// SIMATIC STEP 7 (V5.x) project COB#1&2_CC#2_07_12_2012
// CPU: CPU 315-2 DP
// CPU: CPU 315-2 DP
// program: S7 Program
// program: S7 Program

SYMBOL_TABLE
"MAIN_POWER_DB"	DB 1	DB 1
"HYDRALIC_DB"	DB 2	DB 2
"TRAVEL_DRIVE_DB"	DB 3	DB 3
"CC_BUNKER_GATE_DB"	DB 4	DB 4
"OVEN_CHARGING_DB"	DB 5	DB 5
"TATA_COMMUNICATION_DB"	DB 6	DB 6	// TATA COMMUNIATION DATA BLOCK
"INSTANCE DB FOR FM350"	DB 7	UDT 2	// INSTANCE DB FOR FM350
"08_LID_MECHANISM_DB"	DB 8	DB 8
"LIFTING_PLATFORM_DB"	DB 9	DB 9	// LIFTING PLATFORM DATA BLOCK
"CMD_FROM_TATA"	DB 10	DB 10	// COMMANDS RECEIVED THROUGH PROFIBUS FROM TATA
"FB_TO_TATA"	DB 11	DB 11	// FEEDBACK TO TATA THROUGH PROFIBUS
"DOOR_EXTRACTOR_DB"	DB 12	DB 12	// DOOR EXTRACTOR MECHANISH DATA BLOCK
"DOOR_CLEANER_DB"	DB 13	DB 13	// DOOR CLEANER MECHANISM DATA BLOCK
"JAMB_CLEANER_DB"	DB 14	DB 14	// JAMB CLEANER MECHANISM DATA BLOCK
"WINCC_DB"	DB 15	DB 15
"COAL_SPILLAGE_SYSTEM_DB"	DB 16	DB 16	// COAL SPILLAGE SYSTEM DATA BLOCK
"SCREW_FEEDER_PF"	DB 17	DB 17	// SCREW FEEDER PROFIBUS
"TRAVEL_PROFIBUS"	DB 18	DB 18
"SF_PROFIBUS"	DB 19	DB 19	// SCREW FEEDER PROFIBUS FINAL
"MAIN_POWER"	FC 1	FC 1	// MAIN POWER ON FUNCTION
"CNT2_CTR"	FC 2	FC 2	// Control counter module FM 350-2
"CNT2_WR"	FC 3	FC 3	// Write data records to FM 350-2
"CNT2_RD"	FC 4	FC 4	// Read data records from FM 350-2
"INPUT_MAPPING"	FC 5	FC 5	// INPUT MAPPING OF ALL INPUT
"OUTPUT_MAPPING"	FC 6	FC 6	// OUTPUT MAPPING OF ALL OUTPUT
"HYDRALIC_FUNCTION"	FC 7	FC 7
"TRAVEL_DRIVE"	FC 8	FC 8
"BUNKER_GATE"	FC 9	FC 9
"OVEN_CHARGING_SF"	FC 10	FC 10	// SCREW FEEDERS OPERATION
"LID_1_MECHANISM"	FC 11	FC 11	// LID MECHANISM OF PUSHER SIDE
"PROFIBUS COMMUNICATION"	FC 12	FC 12	// PROFIBUS COMMUNICATION OF DRIVES
"LID_2_MECHANISM"	FC 13	FC 13	// LID MECHANISM OF MIDDLE SIDE
"LID_3_MECHANISM"	FC 14	FC 14	// LID MECHANISM OF COKE SIDE
"TATA_COMMUNICATION"	FC 21	FC 21	// COMMUNICATION WITH TATA THROUGH PROFIBUS
"SCALE"	FC 105	FC 105	// Scaling Values
"UNSCALE"	FC 106	FC 106	// Unscaling Values
"MAIN_PWR_RDY_FOR_ON"	I 0.0	BOOL	// MAIN POWER READY FOR ON
"MAIN_PWR_ON_FB"	I 0.1	BOOL	// MAIN POWER ON FEEDBACK
"CTRL_PWR_ON_FB"	I 0.2	BOOL	// CONTROL POWER ON FEED BACK
"MAIN_PWR_ON_PB"	I 0.3	BOOL	// MAIN POWER ON PUSH BUTTON
"MAIN_PWR_OFF_PB"	I 0.4	BOOL	// MAIN POWER OFF PUSH BUTTON
"LAMP_TEST_PB"	I 0.5	BOOL	// LAMP TEST PUSH BUTTON CONTROL DESK
"ALRM_ACK_PB"	I 0.6	BOOL	// ALARM ACKNOWLEDGE PUSH BUTTON
"TRA_BYPAS_CMD"	I 0.7	BOOL	// TRAVEL BYPASS COMMAND
"LID_MECH_REP_MODE"	I 1.0	BOOL	// LID MECHANISM REPAIR MODE
"LID_MECH_OPER_MODE"	I 1.1	BOOL	// LID MECHANISM OPERATING MODE
"LID_MECH_MAN_MODE"	I 1.2	BOOL	// LID MECHANISM MANUAL MODE
"LID_MECH_AUTO_MODE"	I 1.3	BOOL	// LID MECHANISM AUTO MODE
"HYD_PUMP_1_RDY_FOR_STA"	I 1.4	BOOL	// HYDRAULIC PUMP 1 READY FOR START
"HYD_PUMP_1_RUN_FB"	I 1.5	BOOL	// HYDRAULIC PUMP 1 RUN FEEDBACK
"HYD_PUMP_1_OVRLD_TRIP"	I 1.6	BOOL	// HYDRAULIC PUMP 1 OVERLOAD TRIP
"TRA_AUTO_MAN_SS"	I 1.7	BOOL	// TRAVEL AUTO / MANUAL SELECTOR SWITCH
"HYD_PUMP_2_RDY_FOR_STA"	I 2.0	BOOL	// HYDRAULIC PUMP 2 READY FOR START
"HYD_PUMP_2_RUN_FB"	I 2.1	BOOL	// HYDRAULIC PUMP 2 RUN FEEDBACK
"HYD_PUMP_2_OVRLD_TRIP"	I 2.2	BOOL	// HYDRAULIC PUMP 2 OVERLOAD TRIP
"CIR_PUMP_RDY_FOR_STA"	I 2.3	BOOL	// CIRCULATION PUMP READY FOR START
"CIR_PUMP_ON_FB"	I 2.4	BOOL	// CIRCULATION PUMP RUNNING FEEDBACK
"CIR_PUMP_OVRLD_TRIP"	I 2.5	BOOL	// CIRCULATION PUMP OVERLOAD TRIP
"COOL_FAN_RDY_FOR_STA"	I 2.6	BOOL	// CIRCULATION PUMP READY FOR START
"PROX_MODE_SEL_SF_1"	I 2.7	BOOL	// PROXIMITY MODE SELECTION SCREW FEEDER 1
"COOL_FAN_RUN_FB"	I 3.0	BOOL	// HYDRAULIC COOLER FAN RUN FEEDBACK
"COOL_FAN_OVRLD_TRIP"	I 3.1	BOOL	// HYDRAULIC COOLER FAN OVERLOAD TRIP
"LID_FRAME_CLR_BYBASS"	I 3.2	BOOL	// LID AND FRAME CLEANER BYPASS INPUT
"SPARE_1"	I 3.3	BOOL
"HYD_CD_LCS_SS"	I 3.5	BOOL	// HYDRAULIC PUMP CD/LCS SELECTOR SWITCH
"HYD_PUMP_1_2_SS"	I 3.6	BOOL	// HYDRAULIC PUMP 1 OR 2 SELECTOR SWITCH
"PROX_MODE_SEL_SF_2"	I 3.7	BOOL	// PROXIMITY MODE SELECTION SCREW FEEDER 2
"PUMP_1_STA_PB"	I 4.0	BOOL	// PUMP 1 START PUSH BUTTON
"PUMP_1_STP_PB"	I 4.1	BOOL	// PUMP 1 STOP PUSH BUTTON
"PUMP_2_STA_PB"	I 4.2	BOOL	// PUMP 2 START PUSH BUTTON
"PUMP_2_STP_PB"	I 4.3	BOOL	// PUMP 2 STOP PUSH BUTTON
"EMER_PB_AT_LCS_41"	I 4.4	BOOL	// EMER_PB_AT_LCS 41
"PUMP_1_STA_PB_LCS"	I 4.5	BOOL	// PUMP 1 START PUSH BUTTON AT LCS
"PUMP_1_STP_PB_LCS"	I 4.6	BOOL	// PUMP 1 STOP PUSH BUTTON AT LCS
"PROX_MODE_SEL_SF_3"	I 4.7	BOOL	// PROXIMITY MODE SELECTION SCREW FEEDER 3
"HYD_PUMP_1_2_SS_LCS"	I 5.0	BOOL	// HYDRAULIC PUMP 1 OR 2 SELECTOR SWITCH LCS
"PUMP_2_STA_PB_LCS"	I 5.1	BOOL	// PUMP 2 START PUSH BUTTON AT LCS
"PUMP_2_STP_PB_LCS"	I 5.2	BOOL	// PUMP 2 STOP PUSH BUTTON AT LCS
"CIR_PUMP_STA_PB"	I 5.3	BOOL	// CIRCULATION PUMP START PUSH BUTTON
"CIR_PUMP_STP_PB"	I 5.4	BOOL	// CIRCULATION PUMP STOP PUSH BUTTON
"COOL_FAN_STA_PB"	I 5.5	BOOL	// COOLLER FAN START PUSH BUTTON
"COOL_FAN_STP_PB"	I 5.6	BOOL	// COOLLER FAN STOP PUSH BUTTON
"LAMP_TEST_AT_HYD_LCS"	I 6.0	BOOL	// LAMP TEST PUSH BUTTON AT HYDRALIC LCCS
"ACCUM_STA_PB"	I 6.1	BOOL	// ACCUMULATOR START PUSH BUTTON
"ACCUM_STP_PB"	I 6.2	BOOL	// ACCUMULATOR STOP PUSH BUTTON
"SPARE_2"	I 6.3	BOOL
"SPARE _3"	I 6.4	BOOL
"SHTOFF_VALVE_LINE_1_OPEN"	I 6.5	BOOL	// SHUTOFF VALVE LINE 1 OPEN
"SHTOFF_VALVE_LINE_2_OPEN"	I 6.6	BOOL	// SHUTOFF VALVE LINE 2 OPEN
"LOW_OIL_TEMP"	I 7.0	BOOL	// HYDRALIC LOW OIL TEMPERATURE FROM (THERM)
"HIGH_OIL_TEMP"	I 7.1	BOOL	// HYDRALIC HIGH OIL TEMPERATURE FROM (THERM)
"MAXI_OIL_TEMP"	I 7.2	BOOL	// HYDRALIC MAXI OIL TEMPERATURE FROM (THERM)
"HYD_LO_OIL_LEV"	I 7.3	BOOL	// HYDRALIC LOW OIL LEVEL FLOAT SWITCH
"HYD_MIN_OIL_LEV"	I 7.4	BOOL	// HYDRALIC MINIMUM OIL LEVEL FLOAT SWITCH
"RET_LIN_FILT_CHOKE"	I 7.5	BOOL	// RETURN LINE FILTER CHOKE
"LOW_OIL_PRES_SW"	I 7.6	BOOL	// LOW OIL PRESSURE SWITCH
"RET_LINE_2_FIL_CHK"	I 7.7	BOOL	// RETURN LINE 2 FILTER CHOKE
"HIGH_OIL_PRES"	I 8.0	BOOL	// HIGH OIL PRESSURE SWITCH
"TRA_GRP_1_RDY_FOR_STA"	I 8.1	BOOL	// TRAVEL GROUP MOTOR 1 READY FOR START
"TRA_GRP_1_MTR_RUN_FB"	I 8.2	BOOL	// TRAVEL GROUP MOTOR 1 RUN FEEDBACK
"TRA_MTR_1_OVRLD_TRIP"	I 8.3	BOOL	// TRAVEL MOTOR 1 OVERLOAD TRIP
"TRA_MTR_2_OVRLD_TRIP"	I 8.4	BOOL	// TRAVEL MOTOR 2 OVERLOAD TRIP
"SIR_RDY_FOR_STA"	I 8.5	BOOL	// SIREN READY FOR START
"SIR_RUN_FB"	I 8.6	BOOL	// SIREN RUNNING FEEDBACK
"HOPPER_STP_PB"	I 8.7	BOOL	// HOPPER GATE STOP PUSH BUTTON
"SIR_OVRLD_TRIP"	I 9.0	BOOL	// SIREN OVERLOAD TRIP
"BRK_1_RDY_FOR_STA"	I 9.1	BOOL	// BRAKE 1 READY FOR START
"BRK_1_RUN_FB"	I 9.2	BOOL	// BRAKE 1 RUN FEEDBACK
"TRA_GRP_2_RDY_FOR_STA"	I 9.3	BOOL	// TRAVEL GROUP MOTOR 2 READY FOR START
"TRA_GRP_2_MTR_RUN_FB"	I 9.4	BOOL	// TRAVEL GROUP MOTOR 2 RUN FEEDBACK
"TRA_MTR_3_OVRLD_TRIP"	I 9.5	BOOL	// TRAVEL MOTOR 3 OVERLOAD TRIP
"TRA_MTR_4_OVRLD_TRIP"	I 9.6	BOOL	// TRAVEL MOTOR 4 OVERLOAD TRIP
"BRK_2_RDY_FOR_STA"	I 10.0	BOOL	// BRAKE 2 READY FOR START
"BRK_2_RUN_FB"	I 10.1	BOOL	// BRAKE 2 RUN FEEDBACK
"TRA_JOY_STK_HME_POS"	I 10.2	BOOL	// TRAVEL JOYSTICK HOME POSITION
"TRA_JOY_STK_FWD_POS"	I 10.3	BOOL	// TRAVEL JOYSTICK FORWARD POSITION
"TRA_JOY_STK_REV_POS"	I 10.4	BOOL	// TRAVEL JOYSTICK REVERSE POSITION
"TRA_JOY_STK_DEAD_MAN_PB"	I 10.5	BOOL	// TRAVEL JOYSTICK DEADMAN PUSH BUTTON
"SPARE_4"	I 10.6	BOOL
"TRA_DRV_1_HW_PF_SS"	I 11.0	BOOL	// TRAVEL DRIVE 1 HARDWARE PROFIBUS SELECTOR SWITCH
"TRA_DRV_1_RUN_FB"	I 11.1	BOOL	// TRAVEL DRIVE 1 RUNING FEEDBACK
"TRA_DRV_1_RDY_FOR_STA"	I 11.2	BOOL	// TRAVEL DRIVE 1 READY FOR START
"TRA_DRV_1_TRIP_FB"	I 11.3	BOOL	// TRAVEL DRIVE 1 TRIP FEED BACK
"TRA_DRV_2_HW_PF_SS"	I 11.4	BOOL	// TRAVEL DRIVE 2 HARDWARE PROFIBUS SELECTOR SWITCH
"TRA_DRV_2_RUN_FB"	I 11.5	BOOL	// TRAVEL DRIVE 2 RUNING FEEDBACK
"TRA_DRV_2_RDY_FOR_STA"	I 11.6	BOOL	// TRAVEL DRIVE 2 READY FOR START
"SPARE_5"	I 11.7	BOOL
"TRA_DRV_2_TRIP_FB"	I 12.0	BOOL	// TRAVEL DRIVE 2 TRIP FEED BACK
"LIMIT_SWITCH_END_FWD_FB"	I 12.1	BOOL	// OVER TRAVEL LIMIT SWITCH
"LONG_TRA_SLOW_SPD"	I 12.2	BOOL	// LONG TRAVEL MAKES SLOW SPEED
"LIMIT_SWITCH_END_REV_FB"	I 12.3	BOOL	// LIMIT SWITCH END REVERSE FEED BACK
"SF_1_HW_PF_SS"	I 12.5	BOOL	// SCREW FEEDER 1 HARDWARE/PROFIBUS SELECTOR SWITCH
"SF_1_RDY_FOR_STA"	I 12.6	BOOL	// SCREW FEEDER 1 READY FOR START
"SPARE _6"	I 12.7	BOOL
"SF_1_RUN_FB"	I 13.0	BOOL	// SCREW FEEDER 1 RUNING FEEDBACK
"SF_1_TRIP_FB"	I 13.1	BOOL	// SCREW FEEDER 1 TRIP FEEDBACK
"SF_2_HW_PF_SS"	I 13.2	BOOL	// SCREW FEEDER 2 HARDWARE/PROFIBUS SELECTOR SWITCH
"SF_2_RDY_FOR_STA"	I 13.3	BOOL	// SCREW FEEDER 2 READY FOR START
"SF_2_RUN_FB"	I 13.4	BOOL	// SCREW FEEDER 2 RUNING FEEDBACK
"SF_2_TRIP_FB"	I 13.5	BOOL	// SCREW FEEDER 2 TRIP FEEDBACK
"SF_3_HW_PF_SS"	I 13.6	BOOL	// SCREW FEEDER 3 HARDWARE/PROFIBUS SELECTOR SWITCH
"SPARE_7"	I 13.7	BOOL
"SF_3_RDY_TO_STA"	I 14.0	BOOL	// SCREW FEEDER 3 READY FOR START
"SF_3_RUN_FB"	I 14.1	BOOL	// SCREW FEEDER 2 RUNING FEEDBACK
"SF_3_TRIP_FB"	I 14.2	BOOL	// SCREW FEEDER 3 TRIP FEEDBACK
"SPARE_8"	I 14.3	BOOL
"DC_POWER_PACK1_ON_CMD"	I 14.4	BOOL
"SF _1_STA_PB"	I 14.5	BOOL	// SCREW FEEDER 1 START PUSH BUTTON
"SF_1_STP_PB"	I 14.6	BOOL	// SCREW FEEDER 1 STOP PUSH BUTTON
"SPARE_9"	I 14.7	BOOL
"SF_1_HIGH_SPD_SEL"	I 15.0	BOOL	// SCREW FEEDER 1 HIGH SPEED SELECTION
"SF_1_LOW_SPD_SEL"	I 15.1	BOOL	// SCREW FEEDER 1 LOW SPEED SELECTION
"SF_2_STA_PB"	I 15.2	BOOL	// SCREW FEEDER 2 START PUSH BUTTON
"SF_2_STP_PB"	I 15.3	BOOL	// SCREW FEEDER 2 STOP PUSH BUTTON
"SF_2_HIGH_SPD_SEL"	I 15.4	BOOL	// SCREW FEEDER 2  HIGH SPEED SELECTION
"SF -2 LOW SPEED SELECT"	I 15.5	BOOL	// SCREW FEEDER 2 LOW SPEED SELECTION
"SF_3_STA_PB"	I 15.6	BOOL	// SCREW FEEDER 3 START PUSH BUTTON
"SPARE_10"	I 15.7	BOOL
"SF_3_STP_PB"	I 16.0	BOOL	// SCREW FEEDER 3 STOP PUSH BUTTON
"SF_3_HI_SPD_SEL"	I 16.1	BOOL	// SCREW FEEDER 3 HIGH SPEED SELECTION
"SF_3_LOW_SPD_SEL"	I 16.2	BOOL	// SCREW FEEDER 3 LOW SPEED SELECTION
"LID_LUT_TANK_RDY_FOR_STA"	I 16.3	BOOL	// LID LUTTING TANK READY FOR START
"LID_LUT_TANK_RUN_FB"	I 16.4	BOOL	// LID LUTTING TANK RUN FEEDBACK
"LID_LUT_TANK_OVRLD_TRIP"	I 16.5	BOOL	// LID LUTTING TANK TRIP FEEDBACK
"LID_LUT_TANK_STA_PB"	I 16.6	BOOL	// LID LUTTING TANK START PUSH BUTTON
"SPARE_11"	I 16.7	BOOL
"LID_LUT_TANK_STP_PB"	I 17.0	BOOL	// LID LUTTING TANK STOP PUSH BUTTON
"MAG_ENER_RDY_FOR_START"	I 17.1	BOOL	// MAGNET ENERGISING READY FOR START
"MAG_1_EMER_FB"	I 17.2	BOOL	// MAGNET 1 ENERGISED FEEDBACK
"MAG_2_EMER_FB"	I 17.3	BOOL	// MAGNET 2 ENERGISED FEEDBACK
"MAG_3_EMER_FB"	I 17.4	BOOL	// MAGNET 2 ENERGISED FEEDBACK
"MAG_RUN_FB"	I 17.5	BOOL	// MAGNET RUNNING FEEDBACK
"MAG 1_STA_PB"	I 17.6	BOOL	// MAGNET 1 START PUSH BUTTON
"SPARE_12"	I 17.7	BOOL
"MAG_1_STP_PB"	I 18.0	BOOL	// MAGNET 1 STOP PUSH BUTTON
"MAG_2_STA_PB"	I 18.1	BOOL	// MAGNET 2 START PUSH BUTTON
"MAG_2_STP_PB"	I 18.2	BOOL	// MAGNET 2 STOP PUSH BUTTON
"MAG_3_STA_PB"	I 18.3	BOOL	// MAGNET 2 START PUSH BUTTON
"MAG_3_STP_PB"	I 18.4	BOOL	// MAGNET 3 STOP PUSH BUTTON
"LID_1_AT_MAG_LS"	I 18.5	BOOL	// LID 1 AT MAGNET LIMIT SWITCH
"LID_2_AT_MAG_LS"	I 18.6	BOOL	// LID 2 AT MAGNET LIMIT SWITCH
"SPARE_13"	I 18.7	BOOL
"LID 3_AT_MAG_LS"	I 19.0	BOOL	// LID 3 AT MAGNET LIMIT SWITCH
"LID_1_OSC_MTR_RDY_STA"	I 19.1	BOOL	// LID 1 OSCILLATION MOTOR READY FOR START
"LID_1_OSC_MTR_RUN_FB"	I 19.2	BOOL	// LID 1 OSCILLATION MOTOR RUN FEEDBACK
"LID_1_OSC_MTR_OLR_TRIP"	I 19.3	BOOL	// LID 1 OSCILLATION MOTOR OVERLOAD TRIP
"LID_2_OSC_MTR_RDY_STA"	I 19.4	BOOL	// LID 2 OSCILLATION MOTOR READY FOR START
"LID_2_OSC_MTR_RUN_FB"	I 19.5	BOOL	// LID 2 OSCILLATION MOTOR RUN FEEDBACK
"LID_2_OSC_MTR_OLR_TRIP"	I 19.6	BOOL	// LID 2 OSCILLATION MOTOR OVERLOAD TRIP
"SPARE14"	I 19.7	BOOL
"LID_3_OSC_MTR_RDY_STA"	I 20.0	BOOL	// LID 3 OSCILLATION MOTOR READY FOR START
"LID_3_OSC_MTR_RUN_FB"	I 20.1	BOOL	// LID 3 OSCILLATION MOTOR RUN FEEDBACK
"LID_3_OSC_MTR_OLR_TRIP"	I 20.2	BOOL	// LID 3 OSCILLATION MOTOR OVERLOAD TRIP FEEDBACK
"LID_1_OSC_MTR_STA_PB"	I 20.3	BOOL	// LID 1 OSCILLATION MOTOR START PUSH BUTTON
"LID_1_OSC_MTR_STP_PB"	I 20.4	BOOL	// LID 1 OSCILLATION MOTOR STOP PUSH BUTTON
"LID_2_OSC_MTR_STA_PB"	I 20.5	BOOL	// LID 2 OSCILLATION MOTOR START PUSH BUTTON
"LID 2_OSC_MTR_STOP_PB"	I 20.6	BOOL	// LID 2 OSCILLATION MOTOR STOP PUSH BUTTON
"SPARE_15"	I 20.7	BOOL
"LID_3_OSC_MTR_STA_PB"	I 21.0	BOOL	// LID 3 OSCILLATION MOTOR START PUSH BUTTON
"LID_3_OSC_MTR_STOP_PB"	I 21.1	BOOL	// LID 3 OSCILLATION MOTOR STOP PUSH BUTTON
"LID_FR_CLN_MTR_1_RDY_STA"	I 21.2	BOOL	// LID FRAME CLEANER MOTOR 1 READY FOR START
"LID_FR_CLNR_MTR_1_RUN_FB"	I 21.3	BOOL	// LID FRAME CLEANER MOTOR 1 RUN FEEDBACK
"LID_FR_CLN_MTR_1_OLR"	I 21.4	BOOL	// LID FRAME CLEANER MOTOR 1 OVERLOAD TRIP
"LID_FR_CLN_MT_2_RDY_STA"	I 21.5	BOOL	// LID FRAME CLEANER MOTOR 2 READY FOR START
"LID_FR_CLN_MTR_2_RUN_FB"	I 21.6	BOOL	// LID FRAME CLEANER MOTOR 2 RUN FEEDBACK
"SPARE_16"	I 21.7	BOOL
"LID_FR_CLN_MTR_2_OLR"	I 22.0	BOOL	// LID FRAME CLEANER MOTOR 2 OVERLOAD TRIP
"LID_FR_CLN_MTR_3_RDY_STA"	I 22.1	BOOL	// LID FRAME CLEANER MOTOR 3 READY FOR START
"LID_FR_CLNR_MTR_3_RUN_FB"	I 22.2	BOOL	// LID FRAME CLEANER MOTOR 3 RUN FEEDBACK
"LID_FR_CLN_MTR_3_OLR"	I 22.3	BOOL	// LID FRAME CLEANER MOTOR 3 OVERLOAD TRIP
"LID_FR_CL_MTR_1_STA_PB"	I 22.4	BOOL	// LID 1 FRAME CLEANER MOTOR START PUSH BUTTON
"LID_FR_CLN_MTR_1_STP_PB"	I 22.5	BOOL	// LID 1 FRAME CLEANER MOTOR STOP PUSH BUTTON
"LID_FR_CL_MT_2_STA_PB"	I 22.6	BOOL	// LID 2 FRAME CLEANER MOTOR START PUSH BUTTON
"SPARE_17"	I 22.7	BOOL
"LID_FR_CLN_MTR_2_STP_PB"	I 23.0	BOOL	// LID 2 FRAME CLEANER MOTOR STOP PUSH BUTTON
"LID_FR_CL_MTR_3_STA_PB"	I 23.1	BOOL	// LID 3 FRAME CLEANER MOTOR START PUSH BUTTON
"LID_FR_CLN_MTR_3_STP_PB"	I 23.2	BOOL	// LID 3 FRAME CLEANER MOTOR STOP PUSH BUTTON
"LID_LIFT_1_CA_FWD_STA"	I 23.3	BOOL	// LID LIFTER 1 CARRIAGE FORWARD START PUSH BUTTON
"LID_LIFT_1_CA_RET_STA"	I 23.4	BOOL	// LID LIFTER 1 CARRIAGE RETRACT START PUSH BUTTON
"LID_LIFT_1_VER_DN_STA"	I 23.5	BOOL	// LID LIFTER 1 VERTICAL DOWN START START PUSH BUTTON
"LID_LIFT_1_VER_UP_STA"	I 23.6	BOOL	// LID LIFTER 1 VERTICAL UP START PUSH BUTTON
"SPARE_18"	I 23.7	BOOL
"LID_FR_CLNR_1_DN_STA"	I 24.0	BOOL	// FRAME CLEANER  1 DOWN START PUSH BUTTON
"LID_FR_CLNR_1_UP_STA"	I 24.1	BOOL	// FRAME CLEANER  1 UP START PUSH BUTTON
"TELESCOPE_1_DOWN_STA"	I 24.2	BOOL	// TELESCOPE 1 DOWN START PUSH BUTTON
"TELESCOPE_1_UP_STA"	I 24.3	BOOL	// TELESCOPE 1 UP START PUSH BUTTON
"SLIDE_GATE_1_CLS_STA"	I 24.4	BOOL	// SLIDE GATE 1 CLOSE START PB
"SLIDE_GATE_1_OPN_STA"	I 24.5	BOOL	// SLIDE GATE 1 OPEN START PB
"SPARE_19"	I 24.6	BOOL
"SPARE_20"	I 24.7	BOOL
"LID_LIFT_1_CAR_FWD_LS"	I 25.0	BOOL	// LID LIFTER 1 CARRIAGE FORWARD LIMIT SWITCH
"LID_LIFT_1_CAR_RET_LS"	I 25.1	BOOL	// LID LIFTER 1 CARRIAGE RETRACT LIMIT SWITCH
"LID_LIFT_1_VER_DN_LS"	I 25.2	BOOL	// LID LIFTER 1 VERTICAL DOWN LIMIT SWITCH
"LID_LIFT_1_VER_UP_LS"	I 25.3	BOOL	// LID LIFTER 1 VERTICAL UP LIMIT SWITCH
"LID_LIFT_1_VER_CLN_LS"	I 25.4	BOOL	// LID LIFTER 1 CLEANING LIMIT SWITCH
"LID_FR_CLNR_1_DN_LS"	I 25.5	BOOL	// LID FRAME CLEANER 1 DOWN  LIMIT SWITCH
"LID_FR_CLNR_1_UP_LS"	I 25.6	BOOL	// LID FRAME CLEANER 1 UP  LIMIT SWITCH
"SPARE_21"	I 25.7	BOOL
"TELES_1_DOWN_LS"	I 26.0	BOOL	// TELESCOPE 1 DOWN  LIMIT SWITCH
"TELES_1_UP_LS"	I 26.1	BOOL	// TELESCOPE 1 UP LIMIT SWITCH
"SLIDE_GATE_1_FWD_LS"	I 26.2	BOOL	// SLIDE GATE 1 FORWARD LIMIT SWITCH
"SLIDE_GATE_1_RET_LS"	I 26.3	BOOL	// SLIDE GATE 1 RETRACT LIMIT SWITCH
"LID_LIFT_2_CAR_FWD_STA"	I 26.5	BOOL	// LID LIFTER 2 CARRIAGE FORWARD START PUSH BUTTOM
"LID_LIFT_2_CAR_RET_STA"	I 26.6	BOOL	// LID LIFTER 2 CARRIAGE RETRACT START PUSH BUTTON
"SPARE_22"	I 26.7	BOOL
"LID_LIFT_2_VER_DN_STA"	I 27.0	BOOL	// LID LIFTER 2 VERTICAL DOWN START START PUSH BUTTON
"LID_LIFT_2_VER_UP_STA"	I 27.1	BOOL	// LID LIFTER 2 VERTICAL UP START PUSH BUTTON
"LID_FR_CLNR_2_DN_STA"	I 27.2	BOOL	// FRAME CLEANER  2 DOWN START PUSH BUTTON
"LID_FR_CLNR_2_UP_STA"	I 27.3	BOOL	// FRAME CLEANER  2 UP START PUSH BUTTON
"TELES_2_DOWN_STA"	I 27.4	BOOL	// TELESCOPE 2 DOWN START PUSH BUTTON
"TELES_2_UP_STA"	I 27.5	BOOL	// TELESCOPE 2 UP START PUSH BUTTON
"SLIDE_GATE_2_CLS_STA"	I 27.6	BOOL	// SLIDE GATE 2  CLOSE START PB
"SPARE_23"	I 27.7	BOOL
"SLIDE_GATE_2_OPN_STA"	I 28.0	BOOL	// SLIDE GATE 2 OPEN START PB
"LID_LIFT_2_CARR_FWD_LS"	I 28.2	BOOL	// LID LIFTER 2 CARRIAGE FORWARD LIMIT SWITCH
"LID_LIFT_2_CARR_RET_LS"	I 28.3	BOOL	// LID LIFTER 2 CARRIAGE RETRACT LIMIT SWITCH
"LID_LIFT_2_VER_DN_LS"	I 28.4	BOOL	// LID LIFTER 2 VERTICAL DOWN LIMIT SWITCH
"LID_LIFT_2_VER_UP_LS"	I 28.5	BOOL	// LID LIFTER 2 VERTICAL UP LIMIT SWITCH
"LID_LIFT_2_CLN_POS_LS"	I 28.6	BOOL	// LID LIFTER 1  CLEANING LIMIT SWITCH
"SPARE_24"	I 28.7	BOOL
"LID_FR_CLNR_2_DOWN_LS"	I 29.0	BOOL	// LID FRAME CLEANER 2 DOWN  LIMIT SWITCH
"LID_FR_CLNR 2_UP_LS"	I 29.1	BOOL	// LID FRAME CLEANER 2 UPLIMIT SWITCH
"TELES_2_DOWN_LS"	I 29.2	BOOL	// TELESCOPE 2 DOWN  LIMIT SWITCH
"TELES_2_UP_LS"	I 29.3	BOOL	// TELESCOPE 2 UP  LIMIT SWITCH
"SLIDE_GATE_2_RET_LS"	I 29.4	BOOL	// SLIDE GATE 2 RETRACT LIMIT SWITCH
"SLIDE_GATE_2_FWD_LS"	I 29.5	BOOL	// SLIDE GATE 2 FORWARD LIMIT SWITCH
"SPARE_25"	I 29.7	BOOL
"LID_LIFT_3_CAR_FWD_STA"	I 30.0	BOOL	// LID LIFTER 3 CARRIAGE FORWARD START PUSH BUTTOM
"LID_LIFT_3_CAR_RET_START"	I 30.1	BOOL	// LID LIFTER 3 CARRIAGE RETRACT START PUSH BUTTOM
"LID_LIFT_3_VER_DN_START"	I 30.2	BOOL	// LID LIFTER 3 VERTICAL UP START PUSH BUTTOM
"LID_LIFT_3_VER_UP_START"	I 30.3	BOOL	// LID LIFTER 3 VERTICAL DOWN START PUSH BUTTOM
"LID_FR_CLNR_3_DN_START"	I 30.4	BOOL	// LID FRAME CLEANER 3 DOWN START PUSH BUTTOM
"LID_FR_CLNR 3_UP_START"	I 30.5	BOOL	// LID FRAME CLEANER 3 UPSTART PUSH BUTTOM
"TELES_3_DN_STA"	I 30.6	BOOL	// TELESCOPE 3 DOWN START PUSH BUTTON
"SPARE_26"	I 30.7	BOOL
"TELES_3_UP_STA"	I 31.0	BOOL	// TELESCOPE 3 UP START PUSH BUTTON
"SLIDE_GATE_3_CLS_STA"	I 31.1	BOOL	// SLIDE GATE 3 CLOSE START PB
"SLIDE_GATE_3_OPN_STA"	I 31.2	BOOL	// SLIDE GATE 3 OPEN START PB
"EMER_STP"	I 31.3	BOOL
"LID_LIFT_3_CAR_FWD_LS"	I 31.4	BOOL	// LID LIFTER 3 CARRIAGE FORWARD LIMIT SWITCH
"LID_LIFT_3_CAR_RET_LS"	I 31.5	BOOL	// LID LIFTER 3 CARRIAGE RETRACT LIMIT SWITCH
"LID_LIFT_3_VER_DN_LS"	I 31.6	BOOL	// LID LIFTER 3 VERTICAL DOWN LIMIT SWITCH
"SPARE_27"	I 31.7	BOOL
"LID_LIFT_3_VER_UP_LS"	I 32.0	BOOL	// LID LIFTER 3 VERTICAL UP LIMIT SWITCH
"LID_LIFT_3_VER_CLN_LS"	I 32.1	BOOL	// LID LIFTER 3 CLEANING LIMIT SWITCH
"LID_FR_CLNR_3_DN_LS"	I 32.2	BOOL	// LID FRAME CLEANER 3 DOWN  LIMIT SWITCH
"LID_FR_CLNR_3_UP_LS"	I 32.3	BOOL	// LID FRAME CLEANER 3 UP  LIMIT SWITCH
"TELES_3_DOWN_LS"	I 32.4	BOOL	// TELESCOPE 3 DOWN  LIMIT SWITCH
"TELES_3_UP_LS"	I 32.5	BOOL	// TELESCOPE 3 UP LIMIT SWITCH
"SLIDE_GATE_3_REV_LS"	I 32.6	BOOL	// SLIDE GATE 3 RETRACT LIMIT SWITCH
"SPARE_28"	I 32.7	BOOL
"SLIDE_GATE_3_FWD_LS"	I 33.0	BOOL	// SLIDE GATE 3 FORWARD LIMIT SWITCH
"LCS_EMERGENCY_STP_PB"	I 33.1	BOOL
"BNKR_GATE_MAN_MODE"	I 33.2	BOOL	// BUNKER GATE MANUAL MODE
"BNKR_GATE_REP_MODE"	I 33.3	BOOL	// BUNKER GATE REPAIR MODE
"BNKR_GATE_1_UP_STA_PB"	I 33.4	BOOL	// BUNKER GATE 1 UP START PUSH BUTTON
"BNKR_GATE_1_DN_STA_PB"	I 33.5	BOOL	// BUNKER GATE 1 DOWN START PUSH BUTTON
"BNKR_GATE_1_OPN_STA_PB"	I 33.6	BOOL	// BUNKER GATE 1 OPEN START PUSH BUTTON
"BUKR_GAT OPATION SEMIAUT"	I 33.7	BOOL	// BUNKER GATE SEMI-AUTO MODE
"BNKR_GATE_1_CL_STA_PB"	I 34.0	BOOL	// BUNKER GATE 1 CLOSE START PUSH BUTTON
"BNKR_GATE_2_UP_STA_PB"	I 34.1	BOOL	// BUNKER GATE 2 UP START PUSH BUTTON
"BNKR_GATE_2_DN_STA_PB"	I 34.2	BOOL	// BUNKER GATE 2 DOWN START PUSH BUTTON
"BNKR_GATE_2_OPN_STA_PB"	I 34.3	BOOL	// BUNKER GATE 2 OPEN START PUSH BUTTON
"BNKR_GATE_2_CL_STA_PB"	I 34.4	BOOL	// BUNKER GATE 2 CLOSE START PUSH BUTTON
"BNKR_GATE_3_UP_STA_PB"	I 34.5	BOOL	// BUNKER GATE 3 UP START PUSH BUTTON
"BNKR_GATE_3_DN_STA_PB"	I 34.6	BOOL	// BUNKER GATE 3 DOWN START PUSH BUTTON
"SPARE_29"	I 34.7	BOOL
"BNKR_GATE_3_OPN_STA_PB"	I 35.0	BOOL	// BUNKER GATE 3 OPEN START PUSH BUTTON
"BNKR_GATE_3_CLS_STA_PB"	I 35.1	BOOL	// BUNKER GATE 3 CLOSE START PUSH BUTTON
"BUKR_GATE_COAL_LD_STA_PB"	I 35.2	BOOL	// BUNKER GATE COAL LOAD START PUSH BUTTON
"BUKR_GATE_COAL_LD_STP_PB"	I 35.3	BOOL	// BUNKER GATE COAL LOAD STOP PUSH BUTTON
"BUNKER_GATE_1_UP_LS"	I 35.4	BOOL	// BUNKER GATE 1 UP LIMIT SWITCH
"BUNKER_GATE_1_DN_LS"	I 35.5	BOOL	// BUNKER GATE 1 DOWN LIMIT SWITCH
"BUNKER_GATE_1_OPEN_LS"	I 35.6	BOOL	// BUNKER GATE 1 OPEN LIMIT SWITCH
"TRVL/SCREW SELECTION"	I 35.7	BOOL	// XXXXXXXXXXXXXXXXXXXXXXXXXXXXX
"BUNKER_GATE_1_CLOSE_LS"	I 36.0	BOOL	// BUNKER GATE 1 CLOSE LIMIT SWITCH
"BUNKER_GATE_1_HOME_LS"	I 36.1	BOOL	// BUNKER GATE 1 HOME LIMIT SWITCH
"BUNKER_GATE_2_UP_LS"	I 36.2	BOOL	// BUNKER GATE 2 UP LIMIT SWITCH
"BUNKER_GATE_2_DN_LS"	I 36.3	BOOL	// BUNKER GATE 2 DOWN LIMIT SWITCH
"BUNKER_GATE_2_OPEN_LS"	I 36.4	BOOL	// BUNKER GATE 2 OPEN LIMIT SWITCH
"BUNKER_GATE_2_CLOSE_LS"	I 36.5	BOOL	// BUNKER GATE 2 CLOSE LIMIT SWITCH
"BUNKER_GATE_2_HOME_LS"	I 36.6	BOOL	// BUNKER GATE 2 HOME LIMIT SWITCH
"LID_FR_CLNR_AUTO_MODE"	I 36.7	BOOL
"BUNKER_GATE_3_UP_LS"	I 37.0	BOOL	// BUNKER GATE 3 UP LIMIT SWITCH
"BUNKER_GATE_3_DN_LS"	I 37.1	BOOL	// BUNKER GATE 3 DOWN LIMIT SWITCH
"BUNKER_GATE_3_OPEN_LS"	I 37.2	BOOL	// BUNKER GATE 3 OPEN LIMIT SWITCH
"BUNKER_GATE_3_CLOSE_LS"	I 37.3	BOOL	// BUNKER GATE 3 CLOSE LIMIT SWITCH
"BUNKER_GATE_3_HOME_LS"	I 37.4	BOOL	// BUNKER GATE 3 HOME LIMIT SWITCH
"HOPPER_1_MAXIMUM_LS"	I 37.5	BOOL	// HOPPER 1 MAXIMUM LIMIT SWITCH
"HOPPER_2_MAXIMUM_LS"	I 37.6	BOOL	// HOPPER 2 MAXIMUM LIMIT SWITCH
"BG_1_HM_STA_PB"	I 37.7	BOOL	// BUNKER GATE 3 HOME START PUSH BUTTON
"HOPPER_3_MAXIMUM_LS"	I 38.0	BOOL	// HOPPER 3  MAXIMUM LIMIT SWITCH
"BNKR_GAT_1_UP_STA_PB_LC"	I 38.1	BOOL	// BUNKER GATE 1 UP START PUSH BUTTON LCS
"BNKR_GAT_1_DN_STA_PB_LC"	I 38.2	BOOL	// BUNKER GATE 1 DOWN START PUSH BUTTON LCS
"BNKR_GAT_1_OPN_STA_PB_LC"	I 38.3	BOOL	// BUNKER GATE 1 OPEN START PUSH BUTTON LCS
"BNKR_GAT_1_CLS_STA_PB_LC"	I 38.4	BOOL	// BUNKER GATE 1 CLOSE  START PUSH BUTTON LCS
"BNKR_GAT_1_HME_STA_PB_LC"	I 38.5	BOOL	// BUNKER GATE 1 HOME START PUSH BUTTON LCS
"BNKR_GAT_2_UP_STA_PB_LC"	I 38.6	BOOL	// BUNKER GATE 2 UP START PUSH BUTTON LCS
"BG_2_HME_STA_PB"	I 38.7	BOOL	// BUNKER 2 HOME START PUSH BUTTON
"BNKR_GAT_2_DN_STA_PB_LC"	I 39.0	BOOL	// BUNKER GATE 2 DOWN START PUSH BUTTON LCS
"BNKR_GAT_2_OPN_STA_PB_LC"	I 39.1	BOOL	// BUNKER GATE 2  OPEN START PUSH BUTTON LCS
"BNKR_GAT_2_CLS_STA_PB_LC"	I 39.2	BOOL	// BUNKER GATE 2 CLOSE START PUSH BUTTON LCS
"BNKR_GAT_2_HM_STA_PB_LC"	I 39.3	BOOL	// BUNKER GATE 2 HOME START PUSH BUTTON LCS
"BNKR_GAT_3_UP_STA_PB_LC"	I 39.4	BOOL	// BUNKER GATE 2 UP START PUSH BUTTON LCS
"BNKR_GAT_3_DN_STA_PB_LC"	I 39.5	BOOL	// BUNKER GATE 3 DOWN START PUSH BUTTON LCS
"BNKR_GAT_3_OPN_STA_PB_LC"	I 39.6	BOOL	// BUNKER GATE 3 OPEN START PUSH BUTTON LCS
"BG_3_HM_STA_PB"	I 39.7	BOOL	// BUNKER GATE 3 HOME START PUSH BUTTON
"BNKR_GAT_3_CL_STA_PB_LC"	I 40.0	BOOL	// BUNKER GATE 3 CLOSE START PUSH BUTTON LCS
"BNKR_GAT3_3_HMSTAP_PB_LC"	I 40.1	BOOL	// BUNKER GATE 3 HOME START PUSH BUTTON LCS
"LCS_91_LAMP_TEST"	I 40.2	BOOL	// LCS-91 LAMP TEST PUSH BUTTON
"LCS_91_EMERGENCY_STOP_PB"	I 40.3	BOOL	// LCS-91 EMERGENCY PUSH BUTTON
"DRIVE1 MACRO_FB"	I 40.4	BOOL
"CD_OR_PC_SEL"	I 40.5	BOOL	// CD OR PC SELECTION
"PREPARE_TO_CHARGE"	I 40.6	BOOL	// PREPARE TO CHARGE
"SF_1_PROXI_CNT_INPUT"	I 40.7	BOOL	// SCREW FEEDER 1 PROXIMITY COUNT INPUT
"OVEN_CHARGING_PB"	I 41.0	BOOL	// OVEN CHARING PB FOR AUTO
"FINISH_CHARGING"	I 41.1	BOOL	// FINISH CHARGING PUSH BUTTON
"LID 1_STOP"	I 41.2	BOOL	// LID -1 STOP PUSH BUTTON CD
"LID 2_STOP"	I 41.3	BOOL	// LID -2 STOP PUSH BUTTON CD
"LID 3_STOP"	I 41.4	BOOL	// LID -3 STOP PUSH BUTTON CD
"LEVEL_START_PB"	I 41.5	BOOL
"SIREN_ON_PB"	I 41.6	BOOL	// SIREN ON PUSH BUTTON
"SF_2_PROXI_CNT_INPUT"	I 41.7	BOOL	// SCREW FEEDER 2 PROXIMITY COUNT INPUT
"QUICK_STOP"	I 42.0	BOOL
"AUTO_POSITION_ACKNOWLEGD"	I 42.1	BOOL
"HPALA_LOW_PRESS_START"	I 42.2	BOOL
"HPALA_FIGH PRESS_START"	I 42.3	BOOL
"BIN_GATE_1_PB"	I 42.4	BOOL	// BIN GATE 1 START PUSH BUTTON
"BIN_GATE_2_PB"	I 42.5	BOOL	// BIN GATE 2 START PUSH BUTTON
"BIN_GATE_3_PB"	I 42.6	BOOL	// BIN GATE 3 START PUSH BUTTON
"SF_3_PROXI_CNT_INPUT"	I 42.7	BOOL	// SCREW FEEDER 3 PROXIMITY COUNT INPUT
"CDC_EMERGENCY_STOP"	I 44.4	BOOL	// CDC EMERGENCY STOP
"ALWAYS_OFF"	M 0.0	BOOL	// ALWAYS OFF BIT
"ALWAYS_ON"	M 0.1	BOOL	// ALWAYS ON BIT
"HALF_SECOND_PULSE_TRAIN"	M 0.2	BOOL	// THIS BIT WILL BE ALWAYS ON FOR 500ms AND OFF FOR 500ms
"ONE_SEC_PULSE"	M 0.3	BOOL	// ONE_RAISING EDGE WILL BE GENERATED PER SECOND
"EMERGENCY_PRESSED"	M 0.4	BOOL	// EMERGENCY PUSH BUTTON PRESSED
"PULSE_GENERATION_BIT"	M 0.5	BOOL	// PULSE GENERATION BIT
"LOW_OIL_TEMPE"	M 45.0	BOOL	// LOW OIL TEMPERATURE
"HOP_1_MAX_LS"	M 66.0	BOOL	// HOPPER 1 MAXIMUM LIMIT SWITCH
"HOP_2_MAX_LS"	M 66.2	BOOL	// HOPPER 2 MAXIMUM LIMIT SWITCH
"HOP_3_MAX_LS_SET"	M 66.4	BOOL	// HOPPER 3 MAXIMUM LIMIT SWITCH SET
"PULSE_20"	M 66.5	BOOL
"SCREW_FEEDER_BYPASS"	M 90.0	BOOL
"TEST_BIT"	M 90.1	BOOL
"TEST_BIT_2"	M 90.2	BOOL
"PULSE_1"	M 90.3	BOOL
"PULSE_2"	M 90.4	BOOL
"TRA_PER_IND_BLINK"	M 90.5	BOOL
"ONE_SECOND_PULSE"	M 162.3	BOOL	// ONE RAISING EDGE PULSE PER SECOND
"PROFIBUS_DRIVE_READ_DATA"	MB 108	BYTE
"PROFIBUS_READ_ERROR_D1"	MW 100	INT
"PROFIBUS_WRITE_ERROR_D1"	MW 102	INT
"PROFIBUS_ADDRESS_1"	MW 104	WORD
"PROFIBUS_ADDRESS_2"	MW 106	WORD
"MAIN_PROGRAM"	OB 1	OB 1	// MAIN PROGRAM - CYCLIC EXECUCTION
"CYCL_FLT"	OB 80	OB 80	// Cycle Time Fault
"I/O_FLT1"	OB 82	OB 82	// I/O Point Fault 1
"OBNL_FLT"	OB 85	OB 85	// OB Not Loaded Fault
"RACK_FLT"	OB 86	OB 86	// Loss of Rack Fault
"COMM_FLT"	OB 87	OB 87	// Communication Fault
"COMPLETE RESTART"	OB 100	OB 100	// Complete Restart
"PROG_ERR"	OB 121	OB 121	// Programming Error
"MOD_ERR"	OB 122	OB 122	// Module Access Error
"TRA_JS_IN_VAL"	PIW 256	WORD
"TRA_DRV_JS_SPD_REF"	PIW 258	INT	// TRAVEL DRIVE JOY STICK SPEED REFERENCE
"TRA_DRV_1_SPD_REF"	PQW 256	INT	// TRAVEL DRIVE 1 SPEED REFERENCE
"TRA_DRV_2_SPD_REF"	PQW 258	INT	// TRAVEL DRIVE 2 SPEED REFERENCE
"MAIN PWR START CMD"	Q 0.0	BOOL	// MAIN POWER ON COMMAND
"MAIN PWR READY IND"	Q 0.1	BOOL	// MAIN POWER READY INDICATION
"CONTROL PWR ON INDICATIO"	Q 0.2	BOOL	// CTRL POWER ON INDICATION
"HYD PMP1 ON CMD"	Q 0.3	BOOL	// HYDRAULIC PUMP 1 ON COMMAND
"HYD PMP2 ON CMD"	Q 0.4	BOOL	// HYDRAULIC PUMP 2 ON COMMAND
"CIR PMP ON CMD"	Q 0.5	BOOL	// HYDRAULIC CIRCULATION PUMP ON COMMAND
"COOL FAN ON CMD"	Q 0.6	BOOL	// HYDRAULIC COOLER FAN ON COMMAND
"PRE RELIF VALVE_1 ON CMD"	Q 0.7	BOOL	// PRESSURE RELIEF VALVE ON COMMAND
"SPARE OP 1"	Q 1.0	BOOL
"HYD SYSTEM READY IND"	Q 1.1	BOOL	// HYDRAULIC SYSTEM READY INDICATION
"PUMP1 ON IND CD"	Q 1.2	BOOL	// PUMP 1 ON INDICATION CD
"PUMP2 ON IND CD"	Q 1.3	BOOL	// PUMP 2 ON INDICATION CD
"PUMP1 ON IND LCS"	Q 1.4	BOOL	// PUMP 1 ON INDICATION LCS
"PUMP2 ON IND LCS"	Q 1.5	BOOL	// PUMP 2 ON INDICATION LCS
"CIRC PMP ON IND_LCS"	Q 1.6	BOOL	// CIRCULATION PUMP  ON INDICATION LCS
"SF1 BCD1_3"	Q 1.7	BOOL
"COOL FAN ON IND_LCS"	Q 2.0	BOOL	// COOLER FAN  ON INDICATION LCS
"LOCAL ON IND"	Q 2.1	BOOL	// LOCAL SELECTION ON INDICATION LCS
"HIGH TEMP ON IND_LCS"	Q 2.2	BOOL	// HIGH TEMPERATURE ON INDICATION LCS
"LOWER OIL LVL ON IND_LCS"	Q 2.3	BOOL	// LOWER OIL LEVEL INDICATON LCS
"FILTER CHOHE ON IND_LCS"	Q 2.4	BOOL	// FILTER CHOKE ON INDICATION LCS
"ACCUM_IN_OPER_LCS"	Q 2.5	BOOL	// ACCUMULATOR ON INDICATION LCS
"HEAT_ON_IND_LCS"	Q 2.6	BOOL	// HEATER ON INDICATION LCS
"LOW OIL TEMPERATURE"	Q 2.7	BOOL	// LOWER OIL TEMPERATURE  INDICATON LCS
"TRA GROUP1 ON CMD"	Q 3.0	BOOL
"TRA GROUP2 ON CMD"	Q 3.1	BOOL
"SIREN ON CMD"	Q 3.2	BOOL
"BRAKE ON CMD1"	Q 3.3	BOOL
"BRAKE ON CMD2"	Q 3.4	BOOL
"AUDIO_VISUAL_ALRM_ON_CMD"	Q 3.5	BOOL
"TRA_DRV_FWD"	Q 3.6	BOOL
"TRA_AUD_VIS"	Q 3.7	BOOL	// TRAVEL AUDIO VISUAL SIREN
"TRA_DRV_REV"	Q 4.0	BOOL
"LOGIC I/P 1 TO TR DRIVE"	Q 4.1	BOOL
"LOGIC I/P 2 TO TR DRIVE"	Q 4.2	BOOL
"LOGIC I/P 3 TO TR DRIVE"	Q 4.3	BOOL
"TRA PERMISSION IND"	Q 4.4	BOOL
"TRVL D1 FWD ON CMD"	Q 4.5	BOOL
"TRVL D1 REV ON CMD"	Q 4.6	BOOL
"SPARE 53"	Q 4.7	BOOL
"TRVL D2 FWD ON CMD"	Q 5.0	BOOL
"TRVL D2 REV ON CMD"	Q 5.1	BOOL
"SF -1 HIGH SPEED CMD"	Q 5.2	BOOL
"SF -1 LOW SPEED CMD"	Q 5.3	BOOL
"SF -2 HIGH SPEED CMD"	Q 5.4	BOOL
"SF -2 LOW SPEED CMD"	Q 5.5	BOOL
"SF -3 HIGH SPEED CMD"	Q 5.6	BOOL
"SPARE 52"	Q 5.7	BOOL
"SF -3 LOW SPEED CMD"	Q 6.0	BOOL
"SF -1 ON IND"	Q 6.1	BOOL
"SF -2 ON IND"	Q 6.2	BOOL
"SF -3 ON IND"	Q 6.3	BOOL
"LID LUT TANK ON CMD"	Q 6.4	BOOL
"LID LUT TANK ON IND"	Q 6.5	BOOL
"MAG1 ON CMD"	Q 6.6	BOOL
"BOSTER_CONT_1_ON_CMD"	Q 6.7	BOOL
"MAG2 ON CMD"	Q 7.0	BOOL
"MAG3 ON CMD"	Q 7.1	BOOL
"MAGNET ON CMD"	Q 7.2	BOOL
"MAG1 ON IND"	Q 7.3	BOOL
"MAG2 ON IND"	Q 7.4	BOOL
"MAG3 ON IND"	Q 7.5	BOOL
"LID1 AT MAGNET ON IND"	Q 7.6	BOOL
"BOSTER_CONT_2_ON_CMD"	Q 7.7	BOOL
"LID2 AT MAGNET ON IND"	Q 8.0	BOOL
"LID3 AT MAGNET ON IND"	Q 8.1	BOOL
"LID OSCILLATION1 ON CMD"	Q 8.2	BOOL
"LID OSCILLATION2 ON CMD"	Q 8.3	BOOL
"LID OSCILLATION3 ON CMD"	Q 8.4	BOOL
"LID OSCILLATION1 ON IND"	Q 8.5	BOOL
"LID OSCILLATION2 ON IND"	Q 8.6	BOOL
"BOSTER_CONT_3_ON_CMD"	Q 8.7	BOOL
"LID OSCILLATION3 ON IND"	Q 9.0	BOOL
"LID FR CLEANER1 ON CMD"	Q 9.1	BOOL
"LID FR CLEANER2 ON CMD"	Q 9.2	BOOL
"LID FR CLEANER3 ON CMD"	Q 9.3	BOOL
"LID FR CLEANER1 ON IND"	Q 9.4	BOOL
"LID FR CLEANER2 ON IND"	Q 9.5	BOOL
"LID FR CLEANER3 ON IND"	Q 9.6	BOOL
"SF2 BCD1_4"	Q 9.7	BOOL
"LID LIFT1 CARGE FWD CMD"	Q 10.0	BOOL
"LID LIFT1 CARGE REV CMD"	Q 10.1	BOOL
"LID LIFT1 VERT DWN CMD"	Q 10.2	BOOL
"LID LIFT1 VERT UP CMD"	Q 10.3	BOOL
"LID FR CLEANER1 DOWN CMD"	Q 10.4	BOOL
"LID FR CLEANER1 UP CMD"	Q 10.5	BOOL
"TELESCOPE1 DOWN CMD"	Q 10.6	BOOL
"SF2 BCD1_6"	Q 10.7	BOOL
"TELESCOPE1 UP CMD"	Q 11.0	BOOL
"SLIDE GATE1 CLOSE CMD"	Q 11.1	BOOL
"SLIDE GATE1 OPEN CMD"	Q 11.2	BOOL
"LID LIFT1 CARGE FWD IND"	Q 11.4	BOOL
"LID LIFT1 CARGE REV IND"	Q 11.5	BOOL
"LID LIFT1 VERT DWN IND"	Q 11.6	BOOL
"SF2 BCD1_8"	Q 11.7	BOOL
"LID LIFT1 VERT UP IND"	Q 12.0	BOOL
"LID LIFT1 CLENR POS IND"	Q 12.1	BOOL
"LID FR CLEANER1 DOWN IND"	Q 12.2	BOOL
"LID FR CLEANER1 UP IND"	Q 12.3	BOOL
"TELESCOPE1 DOWN IND"	Q 12.4	BOOL
"TELESCOPE1 UP IND"	Q 12.5	BOOL
"SLIDE GATE1 CLOSE IND"	Q 12.6	BOOL
"SF3 BCD1_1"	Q 12.7	BOOL
"SLIDE GATE1 OPEN IND"	Q 13.0	BOOL
"LID LIFT2 CARGE FWD CMD"	Q 13.2	BOOL
"LID LIFT2 CARGE REV CMD"	Q 13.3	BOOL
"LID LIFT2 VERT DOWN CMD"	Q 13.4	BOOL
"LID LIFT2 VERT UP CMD"	Q 13.5	BOOL
"LID FR CLENR2 DOWN CMD"	Q 13.6	BOOL
"SF3 BCD1_3"	Q 13.7	BOOL
"LID FR CLENR2 UP CMD"	Q 14.0	BOOL
"TELESCOPE2 DOWN CMD"	Q 14.1	BOOL
"TELESCOPE2 UP CMD"	Q 14.2	BOOL
"SLIDE GATE2 CLOSE CMD"	Q 14.3	BOOL
"SLIDE GATE2 OPEN CMD"	Q 14.4	BOOL
"SPARE OUTPUT 6"	Q 14.5	BOOL
"LID LIFT2 CARGE FWD IND"	Q 14.6	BOOL
"SF3 BCD1_4"	Q 14.7	BOOL
"LID LIFT2 CARGE REV IND"	Q 15.0	BOOL
"LID LIFT2 VERT DWN IND"	Q 15.1	BOOL
"LID LIFT2 VERT UP IND"	Q 15.2	BOOL
"LID LIFT2 CLENR POS IND"	Q 15.3	BOOL
"LID FR CLENR2 DOWN IND"	Q 15.4	BOOL
"LID FR CLENR2 UP IND"	Q 15.5	BOOL
"TELESCOPE2 DOWN IND"	Q 15.6	BOOL
"SF3 BCD1_6"	Q 15.7	BOOL
"TELESCOPE2 UP IND"	Q 16.0	BOOL
"SLIDE GATE2 CLOSE IND"	Q 16.1	BOOL
"SLIDE GATE2 OPEN IND"	Q 16.2	BOOL
"LID LIFT3 CARGE FWD CMD"	Q 16.4	BOOL
"LID LIFT3 CARGE REV CMD"	Q 16.5	BOOL
"LID LIFT3 VERT DWN CMD"	Q 16.6	BOOL
"SF3 BCD1_8"	Q 16.7	BOOL
"LID LIFT3 VERT UP CMD"	Q 17.0	BOOL
"LID FR CLENR3 DOWN CMD"	Q 17.1	BOOL
"LID FR CLENR3 UP CMD"	Q 17.2	BOOL
"TELESCOPE3 DOWN CMD"	Q 17.3	BOOL
"TELESCOPE3 UP CMD"	Q 17.4	BOOL
"SLIDE GATE3 CLOSE CMD"	Q 17.5	BOOL
"SLIDE GATE3 OPEN CMD"	Q 17.6	BOOL
"SPARE OUTPUT1"	Q 17.7	BOOL
"LID LIFT3 CARGE FWD IND"	Q 18.1	BOOL
"LID LIFT3 CARGE REV IND"	Q 18.2	BOOL
"LID LIFT3 VERT DWN IND"	Q 18.3	BOOL
"LID LIFT3 VERT UP IND"	Q 18.4	BOOL
"LID LIFT3 CLENR POS IND"	Q 18.5	BOOL
"LID FR CLENR3 DOWN IND"	Q 18.6	BOOL
"SPARE OUTPUT3"	Q 18.7	BOOL
"LID FR CLENR3 UP IND"	Q 19.0	BOOL
"TELESCOPE3 DOWN IND"	Q 19.1	BOOL
"TELESCOPE3 UP IND"	Q 19.2	BOOL
"SLIDE GATE3 CLOSE IND"	Q 19.3	BOOL
"SLIDE GATE3 OPEN IND"	Q 19.4	BOOL
"SPARE OUTPUT7"	Q 19.5	BOOL
"BUNKER GATE1 UP CMD"	Q 19.6	BOOL
"SPARE OUTPUT9"	Q 19.7	BOOL
"BUNKER GATE1 DOWN CMD"	Q 20.0	BOOL
"BUNKER GATE1 OPEN CMD"	Q 20.1	BOOL
"BUNKER GATE1 CLOSE CMD"	Q 20.2	BOOL
"BUNKER GATE2 UP CMD"	Q 20.3	BOOL
"BUNKER GATE2 DOWN CMD"	Q 20.4	BOOL
"BUNKER GATE2 CLOSE CMD"	Q 20.5	BOOL
"BUNKER GATE2 OPEN CMD"	Q 20.6	BOOL
"SPARE OUTPUT17"	Q 20.7	BOOL
"BUNKER GATE3 UP CMD"	Q 21.0	BOOL
"BUNKER GATE3 DOWN CMD"	Q 21.1	BOOL
"BUNKER GATE3 CLOSE CMD"	Q 21.2	BOOL
"BUNKER GATE3 OPEN CMD"	Q 21.3	BOOL
"BUNKER GATE COAL LOD IND"	Q 21.4	BOOL
"LOADING PROGRESS IND"	Q 21.5	BOOL
"BUNKER GATE1 UP IND"	Q 21.6	BOOL
"SPARE OUTPUT18"	Q 21.7	BOOL
"BUNKER GATE1 DOWN IND"	Q 22.0	BOOL
"BUNKER GATE1 OPEN IND"	Q 22.1	BOOL
"BUNKER GATE1 CL0SE IND"	Q 22.2	BOOL
"BUNKER GATE1 HOME IND"	Q 22.3	BOOL
"BUNKER GATE2 UP IND"	Q 22.4	BOOL
"BUNKER GATE2 DN IND"	Q 22.5	BOOL
"BUNKER GATE2 OPEN IND"	Q 22.6	BOOL
"SPARE OUTPUT19"	Q 22.7	BOOL
"BUNKER GATE2 CL0SE IND"	Q 23.0	BOOL
"BUNKER GATE2 HOME IND"	Q 23.1	BOOL
"BUNKER GATE3 UP IND"	Q 23.2	BOOL
"BUNKER GATE3 DOWN IND"	Q 23.3	BOOL
"BUNKER GATE3 OPEN IND"	Q 23.4	BOOL
"BUNKER GATE3 CL0SE IND"	Q 23.5	BOOL
"BUNKER GATE3 HOME IND"	Q 23.6	BOOL
"SPARE OUTPUT20"	Q 23.7	BOOL
"HOPPER1 MAXIMUM IND"	Q 24.0	BOOL
"HOPPER2 MAXIMUM IND"	Q 24.1	BOOL
"HOPPER3 MAXIMUM IND"	Q 24.2	BOOL
"BUNKER GATE 1 UP IND LCS"	Q 24.3	BOOL
"BUNKER GATE 1 DN IND LCS"	Q 24.4	BOOL
"BUNKER GATE 1 OP IND LCS"	Q 24.5	BOOL
"BUNKER GATE 1 CL IND LCS"	Q 24.6	BOOL
"SPARE OUTPUT21"	Q 24.7	BOOL
"BUNKER GATE 1 HM IND LCS"	Q 25.0	BOOL
"BUNKER GATE 2 UP IND LCS"	Q 25.1	BOOL
"BUNKER GATE 2 DN IND LCS"	Q 25.2	BOOL
"BUNKER GATE 2 OP IND LCS"	Q 25.3	BOOL
"BUNKER GATE 2 CL IND LCS"	Q 25.4	BOOL
"BUNKER GATE 2 HM IND LCS"	Q 25.5	BOOL
"BUNKER GATE 3 UP IND LCS"	Q 25.6	BOOL
"SPARE OUTPUT22"	Q 25.7	BOOL
"BUNKER GATE 3 DN IND LCS"	Q 26.0	BOOL
"BUNKER GATE 3 OP IND LCS"	Q 26.1	BOOL
"BUNKER GATE 3 CL IND LCS"	Q 26.2	BOOL
"BUNKER GATE 3 HM IND LCS"	Q 26.3	BOOL
"HOPPER 1 MAXI INDI LCS"	Q 26.4	BOOL
"HOPPER 2 MAXI INDI LCS"	Q 26.5	BOOL
"HOPPER 3 MAXI INDI LCS"	Q 26.6	BOOL
"SPARE OUTPUT25"	Q 26.7	BOOL
"LOCAL SELECTION INDICATI"	Q 27.0	BOOL
"CHARGNG PERMISSION IND"	Q 27.1	BOOL
"CHARGING COMPLETED IND"	Q 27.2	BOOL
"PREPARE TO CHARGE IND"	Q 27.3	BOOL
"OVEN CHARGING IND"	Q 27.4	BOOL
"FINISH CHARGING IND"	Q 27.5	BOOL
"LID 1 PROGRESS IND"	Q 27.6	BOOL
"SPARE OUTPUT29"	Q 27.7	BOOL
"LID 2 PROGRESS IND"	Q 28.0	BOOL
"LID 3 PROGRESS IND"	Q 28.1	BOOL
"LEVEL START"	Q 28.2	BOOL
"HPALA LOP PRESS ON IND"	Q 28.3	BOOL
"PRESSURE RELIEF VALVE 2"	Q 28.4	BOOL
"ACC ON CMD"	Q 28.5	BOOL
"DPRD_DAT"	SFC 14	SFC 14	// Read Consistent Data of a Standard DP Slave
"DPWR_DAT"	SFC 15	SFC 15	// Write Consistent Data to a Standard DP Slave
"BLKMOV"	SFC 20	SFC 20	// Copy Variables
"CREAT_DB"	SFC 22	SFC 22	// Create Data Block
"WR_REC"	SFC 58	SFC 58	// Write Data Record
"RD_REC"	SFC 59	SFC 59	// Read a Data Record
"AUTO_VER_UP_1_DEL"	T 10	TIMER	// VERTICAL UP 1 TIME DELAY AFTER MAGNET OFF
"AUTO_OSC_MTR_ON_OVR"	T 12	TIMER	// AUTO OSCILLATION MOTOR ON TIMER
"BOOSTER_1_OFF_TIMER"	T 13	TIMER	// BOOSTER 1 OFF TIMER
"BOSTER_CONT_2_OFF_TIMER"	T 14	TIMER
"LID_OSC_FB_FLT_TIMER"	T 16	TIMER
"LID_3_OSC_FB_FLT"	T 18	TIMER	// LID OSCILLATION 3 FEEDBACK FLT
"AUTO_OSC_MTR_2_ON_OVR"	T 20	TIMER	// OSCILLATION MOTOR 1 ON OVER
"SF_1_ON_DEL_TIMER"	T 27	TIMER	// SCREW FEEDER 1 ON DELAY TIMER
"SF_2_ON_DEL_TIMER"	T 28	TIMER	// SCREW FEEDER 2 ON DELAY TIMER
"LID_2_VER_UP_TIM_DEL"	T 29	TIMER	// LID 2 VERTICAL UP TIME DELAY AFTER MAGNET OFF
"AUTO_OSC_MTR_3_ON_OVR"	T 30	TIMER	// AUTO OSCILLATION MOTOR 3  ON OVER
"LID_3_VER_UP_TIM_DEL"	T 31	TIMER	// LID 3 VERTICAL UP DELAY AFTER MAGNET OFF
"LID_FR_CLN_MTR_1_OFF_TIM"	T 32	TIMER	// LID FRAME CLEANER MOTOR 1 OFF TIMER
"LID_FRM_CLNR_UP_DEL_TIM"	T 33	TIMER	// LID FRAME CLEANER UP DELAY TIMER
"LID_FRM_CLN_2_UP_DEL_TIM"	T 34	TIMER	// LID FRAME CLEANER 2 MOTOR OFF TIMER
"LID_FRM_CLN_2_STOP_TIM"	T 35	TIMER
"LID_FRM_CLN_UP_DEL_TIM"	T 36	TIMER	// LID FRAME CLEANER UP DELAY TIMER
"LID_FR_CLN_MTR_3_OFF_TIM"	T 37	TIMER	// LID FRAME CLEANER MOTOR 3 OFF TIMER
"BG_1_MAX_LS_CLS_TIM"	T 38	TIMER	// BUNKER GATE 1 MAXIMUM LIMIT SWITCH REACHED
"BG_2_MAX_LS_CLS_TIM"	T 39	TIMER	// BUNKER GATE 2  MAXIMUM LIMIT SWITCH REACHED
"BG_3_MAX_LS_CLS_TIM"	T 40	TIMER	// BUNKER GATE 3  MAXIMUM LIMIT SWITCH REACHED
"PREPARE_CHARGE"	UDT 1	UDT 1
"SCREW_FEEDER"	UDT 2	UDT 2
"FINISH_CHARGE"	UDT 3	UDT 3
"SCREW_FEEDER_SP"	VAT 1		// SCREW FEEDER SET POINTS
"VAT_2"	VAT 2		// OUTPUT_LIST
"VAT_32"	VAT 3	
"PUSHER_RAM_ENCODER"	VAT 4	
"DE_CTRL_SEL_FORCING"	VAT 5	
END_SYMBOL_TABLE

TYPE "PREPARE_CHARGE"	// UDT 1
VERSION : 0.1
  STRUCT
   STEP1 : BOOL ;	//LID LIFTER CAR TRAVEL FWD OVER
   STEP2 : BOOL ;	//LID LIFTER VERT DOWN OVER
   STEP3 : BOOL ;	//LID MAGNET ON FB
   STEP4 : BOOL ;	//LID OSC MOTOR OPRN OVER
   STEP5 : BOOL ;	//LID LIFTER VERT UP OVER
   STEP6 : BOOL ;	//LID LIFTER CAR TRAVEL REV OVER
   STEP7 : BOOL ;	//LID FRAME CLEANER DOWN OVER
   STEP8 : BOOL ;	//LID LIFTER CAR TRAVEL FWD OVER
   STEP9 : BOOL ;	//LID LIFTER VERT DOWN FOR CLN POS OVER
   STEP10 : BOOL ;	//LID CLEANER MOTOR OPRN OVER
   STEP11 : BOOL ;	//LID LIFTER VERT UP FROM CLN POS OVER
   STEP12 : BOOL ;	//LID LIFTER CAR TRAVEL REV OVER
   STEP13 : BOOL ;	//LID FRAME CLEANER UP OVER
   STEP14 : BOOL ;	//TELESCOPE DOWN OVER
   STEP15 : BOOL ;	//LID CLEANER BYPASS ENABLED
   STEP16 : BOOL ;	//LID OSC MOTOR TIME OVER
   STEP17 : BOOL ;	//LID CLEANER MOTOR TIME OVER
   STEP19 : BOOL ;	//PREPARE CHARGE OPERATION COMPLETED
   POS : BOOL ;	//POSITIVE PULSE
   INWORD1 : INT ;	//LID OSC MOTOR TIME MONITOR
   INWORD2 : INT ;	//LID CLEANER MOTOR TIME MONITOR
   INWORD3 : INT ;	//PREPARE CHARGE OPERATION COMPLETION MONITOR
   INWORD4 : DINT ;	//RESERVED BIT FOR PREPARE CHARGE OPRN
  END_STRUCT ;	
END_TYPE

TYPE "SCREW_FEEDER"	// UDT 2
VERSION : 1.0
  STRUCT
   JOB_WR : STRUCT 	// write commands
    NO : BYTE ;	// number
    BUSY : BOOL ;	// job in working
    DONE : BOOL ;	// job is done
    IMPOSS : BOOL ;	// job impossible
    UNKOWN : BOOL ;	// job unkown
   END_STRUCT ;
   JOB_RD : STRUCT 	// read commands
    NO : BYTE ;	// number
    BUSY : BOOL ;	// job in working
    DONE : BOOL ;	// job is done
    IMPOSS : BOOL ;	// job impossible
    UNKOWN : BOOL ;	// job unkown
   END_STRUCT ;
   RESERV_0 : ARRAY  [1 .. 3 ] OF WORD  := 3 (W#16#0) ;	// reserved
   RESERV_1 : WORD ;	// reserved
   MOD_ADR : WORD ;	// module address
   CH_ADR : DWORD ;	// channel address
   DS_OFFS : BYTE ;	// data block offset
   RESERV_2 : BYTE ;	// reserved
   CONTROL_SIGNALS : STRUCT 	// control signals
    BIT0_0 : BOOL ;	// reserved
    BIT0_1 : BOOL ;	// reserved
    BIT0_2 : BOOL ;	// reserved
    BIT0_3 : BOOL ;	// reserved
    BIT0_4 : BOOL ;	// reserved
    BIT0_5 : BOOL ;	// reserved
    BIT0_6 : BOOL ;	// reserved
    BIT0_7 : BOOL ;	// reserved
    CTRL_DQ0 : BOOL ;	// control digital output DQ0
    CTRL_DQ1 : BOOL ;	// control digital output DQ1
    CTRL_DQ2 : BOOL ;	// control digital output DQ2
    CTRL_DQ3 : BOOL ;	// control digital output DQ3
    CTRL_DQ4 : BOOL ;	// control digital output DQ4
    CTRL_DQ5 : BOOL ;	// control digital output DQ5
    CTRL_DQ6 : BOOL ;	// control digital output DQ6
    CTRL_DQ7 : BOOL ;	// control digital output DQ7
    SET_DQ0 : BOOL ;	// set digital output DQ0
    SET_DQ1 : BOOL ;	// set digital output DQ1
    SET_DQ2 : BOOL ;	// set digital output DQ2
    SET_DQ3 : BOOL ;	// set digital output DQ3
    SET_DQ4 : BOOL ;	// set digital output DQ4
    SET_DQ5 : BOOL ;	// set digital output DQ5
    SET_DQ6 : BOOL ;	// set digital output DQ6
    SET_DQ7 : BOOL ;	// set digital output DQ7
    SW_GATE0 : BOOL ;	// software gate 0
    SW_GATE1 : BOOL ;	// software gate 1
    SW_GATE2 : BOOL ;	// software gate 2
    SW_GATE3 : BOOL ;	// software gate 3
    SW_GATE4 : BOOL ;	// software gate 4
    SW_GATE5 : BOOL ;	// software gate 5
    SW_GATE6 : BOOL ;	// software gate 6
    SW_GATE7 : BOOL ;	// software gate 7
    CTRL_DWORD1 : DWORD ;	// reserved
    CTRL_DWORD2 : DWORD ;	// reserved
    CTRL_DWORD3 : DWORD ;	// reserved
   END_STRUCT ;
   CHECKBACK_SIGNALS : STRUCT 	// checkback signals
    BIT0_0 : BOOL ;	// reserved
    STS_TFB : BOOL ;	// status test free bit
    BIT0_2 : BOOL ;	// reserved
    BIT0_3 : BOOL ;	// reserved
    DATA_ERR : BOOL ;	// data error bit
    BIT0_5 : BOOL ;	// reserved
    BIT0_6 : BOOL ;	// reserved
    PARA : BOOL ;	// module parametrized
    STS_CMP0 : BOOL ;	// status compare event 0
    STS_CMP1 : BOOL ;	// status compare event 1
    STS_CMP2 : BOOL ;	// status compare event 2
    STS_CMP3 : BOOL ;	// status compare event 3
    STS_CMP4 : BOOL ;	// status compare event 4
    STS_CMP5 : BOOL ;	// status compare event 5
    STS_CMP6 : BOOL ;	// status compare event 6
    STS_CMP7 : BOOL ;	// status compare event 7
    STS_UFLW0 : BOOL ;	// status counter 0 passed the underflow value
    STS_UFLW1 : BOOL ;	// status counter 1 passed the underflow value
    STS_UFLW2 : BOOL ;	// status counter 2 passed the underflow value
    STS_UFLW3 : BOOL ;	// status counter 3 passed the underflow value
    STS_UFLW4 : BOOL ;	// status counter 4 passed the underflow value
    STS_UFLW5 : BOOL ;	// status counter 5 passed the underflow value
    STS_UFLW6 : BOOL ;	// status counter 6 passed the underflow value
    STS_UFLW7 : BOOL ;	// status counter 7 passed the underflow value
    STS_OFLW0 : BOOL ;	// status counter 0 passed the overflow value
    STS_OFLW1 : BOOL ;	// status counter 1 passed the overflow value
    STS_OFLW2 : BOOL ;	// status counter 2 passed the overflow value
    STS_OFLW3 : BOOL ;	// status counter 3 passed the overflow value
    STS_OFLW4 : BOOL ;	// status counter 4 passed the overflow value
    STS_OFLW5 : BOOL ;	// status counter 5 passed the overflow value
    STS_OFLW6 : BOOL ;	// status counter 6 passed the overflow value
    STS_OFLW7 : BOOL ;	// status counter 7 passed the overflow value
    STS_DIR0 : BOOL ;	// status counter 0 direction
    STS_DIR1 : BOOL ;	// status counter 1 direction
    STS_DIR2 : BOOL ;	// status counter 2 direction
    STS_DIR3 : BOOL ;	// status counter 3 direction
    STS_DIR4 : BOOL ;	// status counter 4 direction
    STS_DIR5 : BOOL ;	// status counter 5 direction
    STS_DIR6 : BOOL ;	// status counter 6 direction
    STS_DIR7 : BOOL ;	// status counter 7 direction
    STS_DI0 : BOOL ;	// status of the digital input 0
    STS_DI1 : BOOL ;	// status of the digital input 1
    STS_DI2 : BOOL ;	// status of the digital input 2
    STS_DI3 : BOOL ;	// status of the digital input 3
    STS_DI4 : BOOL ;	// status of the digital input 4
    STS_DI5 : BOOL ;	// status of the digital input 5
    STS_DI6 : BOOL ;	// status of the digital input 6
    STS_DI7 : BOOL ;	// status of the digital input 7
    STS_DQ0 : BOOL ;	// status of the digital output 0
    STS_DQ1 : BOOL ;	// status of the digital output 1
    STS_DQ2 : BOOL ;	// status of the digital output 2
    STS_DQ3 : BOOL ;	// status of the digital output 3
    STS_DQ4 : BOOL ;	// status of the digital output 4
    STS_DQ5 : BOOL ;	// status of the digital output 5
    STS_DQ6 : BOOL ;	// status of the digital output 6
    STS_DQ7 : BOOL ;	// status of the digital output 7
    STS_GATE0 : BOOL ;	// status of the internal gate 0
    STS_GATE1 : BOOL ;	// status of the internal gate 1
    STS_GATE2 : BOOL ;	// status of the internal gate 2
    STS_GATE3 : BOOL ;	// status of the internal gate 3
    STS_GATE4 : BOOL ;	// status of the internal gate 4
    STS_GATE5 : BOOL ;	// status of the internal gate 5
    STS_GATE6 : BOOL ;	// status of the internal gate 6
    STS_GATE7 : BOOL ;	// status of the internal gate 7
    USER_STAT_WORD0 : WORD ;	// user specific status
    USER_STAT_WORD1 : WORD ;	// user specific status
    USER_STAT_WORD2 : WORD ;	// user specific status
    USER_STAT_WORD3 : WORD ;	// user specific status
   END_STRUCT ;
   LOAD_VAL0 : DINT ;	// load value counter 0
   LOAD_VAL1 : DINT ;	// load value counter 1
   LOAD_VAL2 : DINT ;	// load value counter 2
   LOAD_VAL3 : DINT ;	// load value counter 3
   LOAD_VAL4 : DINT ;	// load value counter 4
   LOAD_VAL5 : DINT ;	// load value counter 5
   LOAD_VAL6 : DINT ;	// load value counter 6
   LOAD_VAL7 : DINT ;	// load value counter 7
   LOAD_PREPARE_VAL0 : DINT ;	// load prepare value counter 0
   LOAD_PREPARE_VAL1 : DINT ;	// load prepare value counter 1
   LOAD_PREPARE_VAL2 : DINT ;	// load prepare value counter 2
   LOAD_PREPARE_VAL3 : DINT ;	// load prepare value counter 3
   LOAD_PREPARE_VAL4 : DINT ;	// load prepare value counter 4
   LOAD_PREPARE_VAL5 : DINT ;	// load prepare value counter 5
   LOAD_PREPARE_VAL6 : DINT ;	// load prepare value counter 6
   LOAD_PREPARE_VAL7 : DINT ;	// load prepare value counter 7
   CMP_VAL0 : DINT ;	// comparator value 0
   CMP_VAL1 : DINT ;	// comparator value 1
   CMP_VAL2 : DINT ;	// comparator value 2
   CMP_VAL3 : DINT ;	// comparator value 3
   CMP_VAL4 : DINT ;	// comparator value 4
   CMP_VAL5 : DINT ;	// comparator value 5
   CMP_VAL6 : DINT ;	// comparator value 6
   CMP_VAL7 : DINT ;	// comparator value 7
   ACT_CNTV0 : DINT ;	// actual counter value 0
   ACT_MSRV0 : DINT ;	// act. measurement value 0
   ACT_CNTV1 : DINT ;	// actual counter value 1
   ACT_MSRV1 : DINT ;	// act. measurement value 1
   ACT_CNTV2 : DINT ;	// actual counter value 2
   ACT_MSRV2 : DINT ;	// act. measurement value 2
   ACT_CNTV3 : DINT ;	// actual counter value 3
   ACT_MSRV3 : DINT ;	// act. measurement value 3
   ACT_CNTV4 : DINT ;	// actual counter value 4
   ACT_MSRV4 : DINT ;	// act. measurement value 4
   ACT_CNTV5 : DINT ;	// actual counter value 5
   ACT_MSRV5 : DINT ;	// act. measurement value 5
   ACT_CNTV6 : DINT ;	// actual counter value 6
   ACT_MSRV6 : DINT ;	// act. measurement value 6
   ACT_CNTV7 : DINT ;	// actual counter value 7
   ACT_MSRV7 : DINT ;	// act. measurement value 7
   DIAGNOSTIC_INT_INFO : STRUCT 	// diagnostic int. information
    BYTE0 : BYTE ;	// byte 0
    BYTE1 : BYTE ;	// byte 1
    BYTE2 : BYTE ;	// byte 2
    BYTE3 : BYTE ;	// byte 3
    BYTE4 : BYTE ;	// channel type info
    BYTE5 : BYTE ;	// channel info length
    BYTE6 : BYTE ;	// number of channels
    BYTE7 : BYTE ;	// channel error vector
    BYTE8 : BYTE ;	// error counter 0
    BYTE9 : BYTE ;	// error counter 1
    BYTE10 : BYTE ;	// error counter 2
    BYTE11 : BYTE ;	// error counter 3
    BYTE12 : BYTE ;	// error counter 4
    BYTE13 : BYTE ;	// error counter 5
    BYTE14 : BYTE ;	// error counter 6
    BYTE15 : BYTE ;	// error counter 7
   END_STRUCT ;
  END_STRUCT ;	
END_TYPE

TYPE "FINISH_CHARGE"	// UDT 3
VERSION : 0.1
  STRUCT
   POS1 : BOOL ;	//POSITIVE PULSE
   STEP_F1 : BOOL ;	//TELESCOPE UP OVER
   STEP_F2 : BOOL ;	//LID LIFTER CAR TRAVEL FWD OVER
   STEP_F3 : BOOL ;	//LID LIFTER VERT DOWN OVER
   STEP_F4 : BOOL ;	//LID MAGNET OFF COMPLETED
   STEP_F5 : BOOL ;	//LID LIFTER VERT UP OVER
   STEP_F6 : BOOL ;	//LID LIFTER CAR TRAVEL REV OVER
   STEP_F7 : BOOL ;	//FINISH CHARGE OPERATION OVER
   IN_WORD5 : INT ;	//FINISH CHARGE OPERATION COMPLETION MONITOR
   IN_WORD6 : INT ;	//RESERVED BIT FOR FINISH TO CHARGE OPRN
  END_STRUCT ;	
END_TYPE

FUNCTION "MAIN_POWER" : VOID	// FC 1
AUTHOR : Arun
VERSION : 0.1
BEGIN
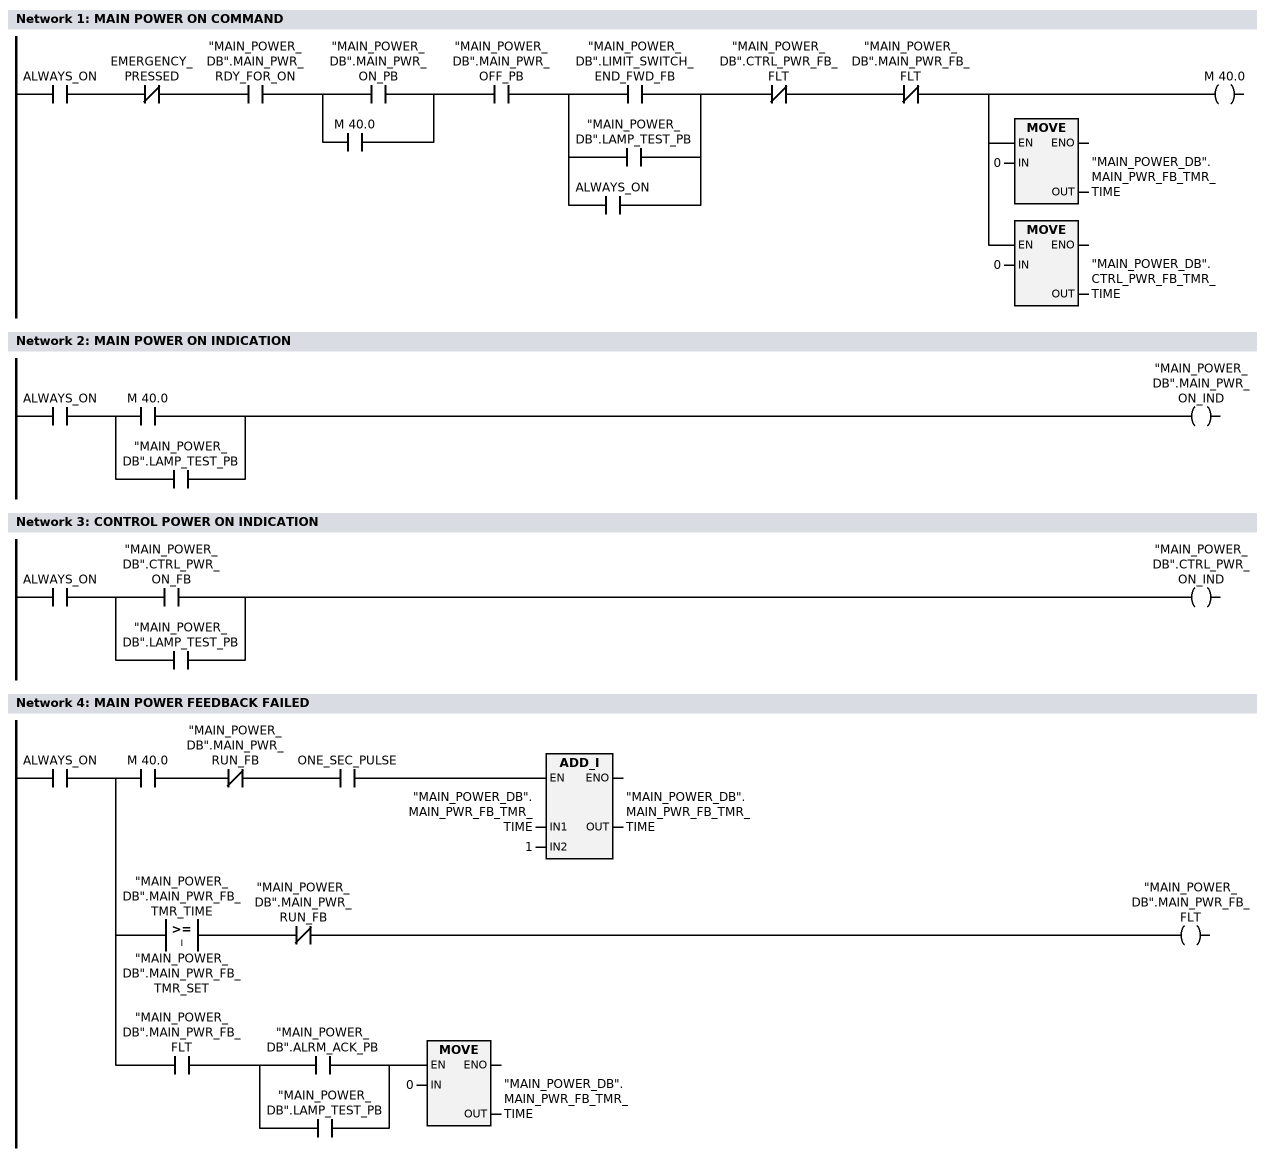
NETWORK
TITLE = MAIN POWER ON COMMAND
      A     "ALWAYS_ON";
      AN    "EMERGENCY_PRESSED";
      A     "MAIN_POWER_DB".MAIN_PWR_RDY_FOR_ON;
      A(;
      O     "MAIN_POWER_DB".MAIN_PWR_ON_PB;
      O     M 40.0;
      );
      A     "MAIN_POWER_DB".MAIN_PWR_OFF_PB;
      A(;
      O     "MAIN_POWER_DB".LIMIT_SWITCH_END_FWD_FB;
      O     "MAIN_POWER_DB".LAMP_TEST_PB;
      O     "ALWAYS_ON";
      );
      AN    "MAIN_POWER_DB".CTRL_PWR_FB_FLT;
      AN    "MAIN_POWER_DB".MAIN_PWR_FB_FLT;
      =     L 0.0;
      A     L 0.0;
      BLD   102;
      =     M 40.0;
      A     L 0.0;
      JNB   _001;
      L     0;
      T     "MAIN_POWER_DB".MAIN_PWR_FB_TMR_TIME;
_001: NOP   0;
      A     L 0.0;
      JNB   _002;
      L     0;
      T     "MAIN_POWER_DB".CTRL_PWR_FB_TMR_TIME;
_002: NOP   0;
NETWORK
TITLE = MAIN POWER ON INDICATION 
      A     "ALWAYS_ON";
      A(;
      O     M 40.0;
      O     "MAIN_POWER_DB".LAMP_TEST_PB;
      );
      =     "MAIN_POWER_DB".MAIN_PWR_ON_IND;
NETWORK
TITLE = CONTROL POWER ON INDICATION
      A     "ALWAYS_ON";
      A(;
      O     "MAIN_POWER_DB".CTRL_PWR_ON_FB;
      O     "MAIN_POWER_DB".LAMP_TEST_PB;
      );
      =     "MAIN_POWER_DB".CTRL_PWR_ON_IND;
NETWORK
TITLE = MAIN POWER FEEDBACK FAILED
      A     "ALWAYS_ON";
      =     L 0.0;
      A     L 0.0;
      A     M 40.0;
      AN    "MAIN_POWER_DB".MAIN_PWR_RUN_FB;
      A     "ONE_SEC_PULSE";
      JNB   _003;
      L     "MAIN_POWER_DB".MAIN_PWR_FB_TMR_TIME;
      L     1;
      +I;
      T     "MAIN_POWER_DB".MAIN_PWR_FB_TMR_TIME;
_003: NOP   0;
      A     L 0.0;
      A(;
      L     "MAIN_POWER_DB".MAIN_PWR_FB_TMR_TIME;
      L     "MAIN_POWER_DB".MAIN_PWR_FB_TMR_SET;
      >=I;
      );
      AN    "MAIN_POWER_DB".MAIN_PWR_RUN_FB;
      =     "MAIN_POWER_DB".MAIN_PWR_FB_FLT;
      A     L 0.0;
      A     "MAIN_POWER_DB".MAIN_PWR_FB_FLT;
      A(;
      O     "MAIN_POWER_DB".ALRM_ACK_PB;
      O     "MAIN_POWER_DB".LAMP_TEST_PB;
      );
      JNB   _004;
      L     0;
      T     "MAIN_POWER_DB".MAIN_PWR_FB_TMR_TIME;
_004: NOP   0;
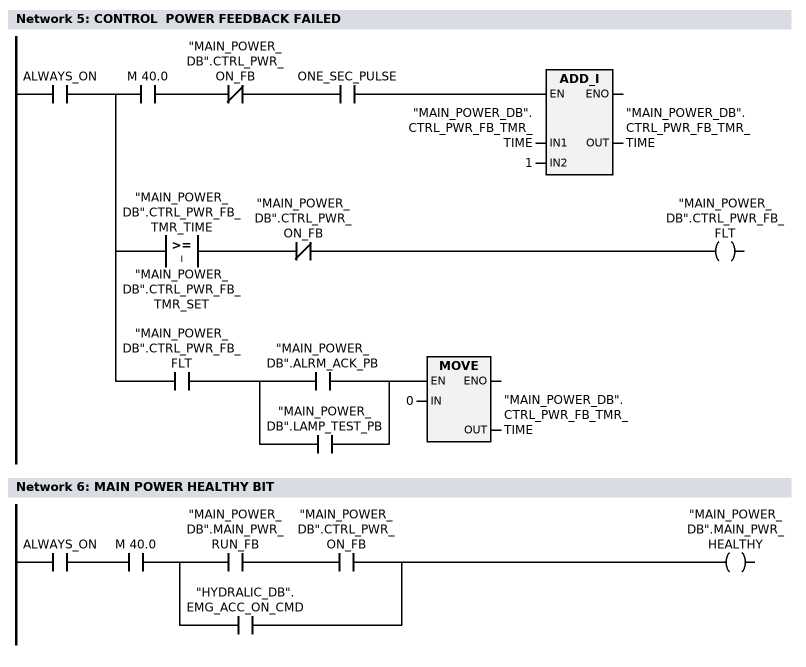
NETWORK
TITLE = CONTROL  POWER FEEDBACK FAILED
      A     "ALWAYS_ON";
      =     L 0.0;
      A     L 0.0;
      A     M 40.0;
      AN    "MAIN_POWER_DB".CTRL_PWR_ON_FB;
      A     "ONE_SEC_PULSE";
      JNB   _005;
      L     "MAIN_POWER_DB".CTRL_PWR_FB_TMR_TIME;
      L     1;
      +I;
      T     "MAIN_POWER_DB".CTRL_PWR_FB_TMR_TIME;
_005: NOP   0;
      A     L 0.0;
      A(;
      L     "MAIN_POWER_DB".CTRL_PWR_FB_TMR_TIME;
      L     "MAIN_POWER_DB".CTRL_PWR_FB_TMR_SET;
      >=I;
      );
      AN    "MAIN_POWER_DB".CTRL_PWR_ON_FB;
      =     "MAIN_POWER_DB".CTRL_PWR_FB_FLT;
      A     L 0.0;
      A     "MAIN_POWER_DB".CTRL_PWR_FB_FLT;
      A(;
      O     "MAIN_POWER_DB".ALRM_ACK_PB;
      O     "MAIN_POWER_DB".LAMP_TEST_PB;
      );
      JNB   _006;
      L     0;
      T     "MAIN_POWER_DB".CTRL_PWR_FB_TMR_TIME;
_006: NOP   0;
NETWORK
TITLE = MAIN POWER HEALTHY BIT
      A     "ALWAYS_ON";
      A     M 40.0;
      A(;
      A     "MAIN_POWER_DB".MAIN_PWR_RUN_FB;
      A     "MAIN_POWER_DB".CTRL_PWR_ON_FB;
      O     "HYDRALIC_DB".EMG_ACC_ON_CMD;
      );
      =     "MAIN_POWER_DB".MAIN_PWR_HEALTHY;
END_FUNCTION

// FC 2: know-how protected block, not included

// FC 3: know-how protected block, not included

// FC 4: know-how protected block, not included

FUNCTION "INPUT_MAPPING" : VOID	// FC 5
AUTHOR : Arun_Ram
VERSION : 0.1
BEGIN
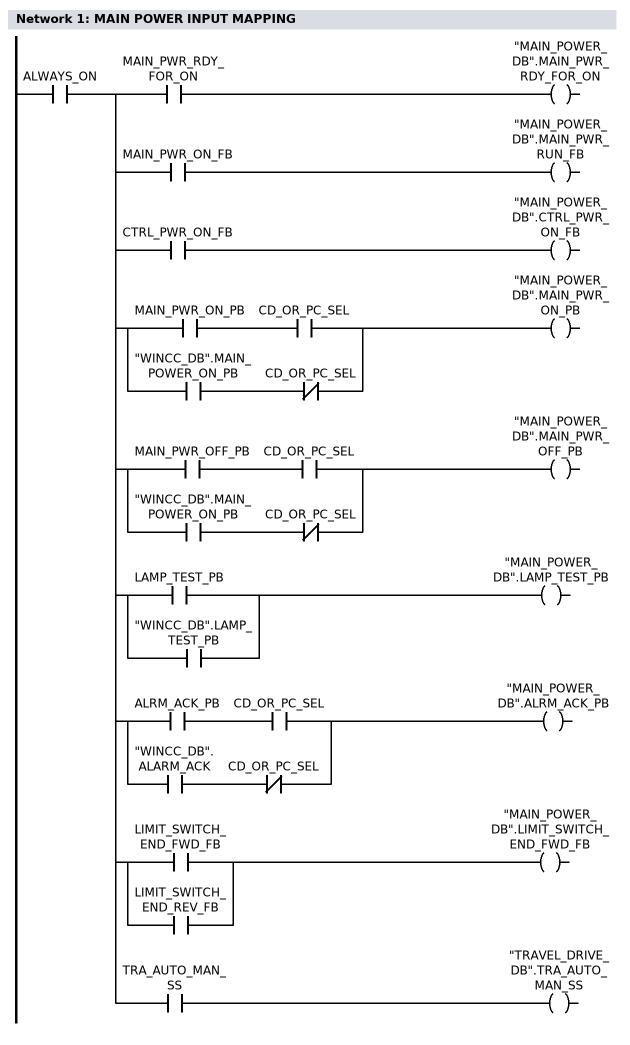
NETWORK
TITLE = MAIN POWER INPUT MAPPING
      A     "ALWAYS_ON";
      =     L 0.0;
      A     L 0.0;
      A     "MAIN_PWR_RDY_FOR_ON";
      =     "MAIN_POWER_DB".MAIN_PWR_RDY_FOR_ON;
      A     L 0.0;
      A     "MAIN_PWR_ON_FB";
      =     "MAIN_POWER_DB".MAIN_PWR_RUN_FB;
      A     L 0.0;
      A     "CTRL_PWR_ON_FB";
      =     "MAIN_POWER_DB".CTRL_PWR_ON_FB;
      A     L 0.0;
      A(;
      A     "MAIN_PWR_ON_PB";
      A     "CD_OR_PC_SEL";
      O;
      A     "WINCC_DB".MAIN_POWER_ON_PB;
      AN    "CD_OR_PC_SEL";
      );
      =     "MAIN_POWER_DB".MAIN_PWR_ON_PB;
      A     L 0.0;
      A(;
      A     "MAIN_PWR_OFF_PB";
      A     "CD_OR_PC_SEL";
      O;
      A     "WINCC_DB".MAIN_POWER_ON_PB;
      AN    "CD_OR_PC_SEL";
      );
      =     "MAIN_POWER_DB".MAIN_PWR_OFF_PB;
      A     L 0.0;
      A(;
      O     "LAMP_TEST_PB";
      O     "WINCC_DB".LAMP_TEST_PB;
      );
      =     "MAIN_POWER_DB".LAMP_TEST_PB;
      A     L 0.0;
      A(;
      A     "ALRM_ACK_PB";
      A     "CD_OR_PC_SEL";
      O;
      A     "WINCC_DB".ALARM_ACK;
      AN    "CD_OR_PC_SEL";
      );
      =     "MAIN_POWER_DB".ALRM_ACK_PB;
      A     L 0.0;
      A(;
      O     "LIMIT_SWITCH_END_FWD_FB";
      O     "LIMIT_SWITCH_END_REV_FB";
      );
      =     "MAIN_POWER_DB".LIMIT_SWITCH_END_FWD_FB;
      A     L 0.0;
      A     "TRA_AUTO_MAN_SS";
      =     "TRAVEL_DRIVE_DB".TRA_AUTO_MAN_SS;
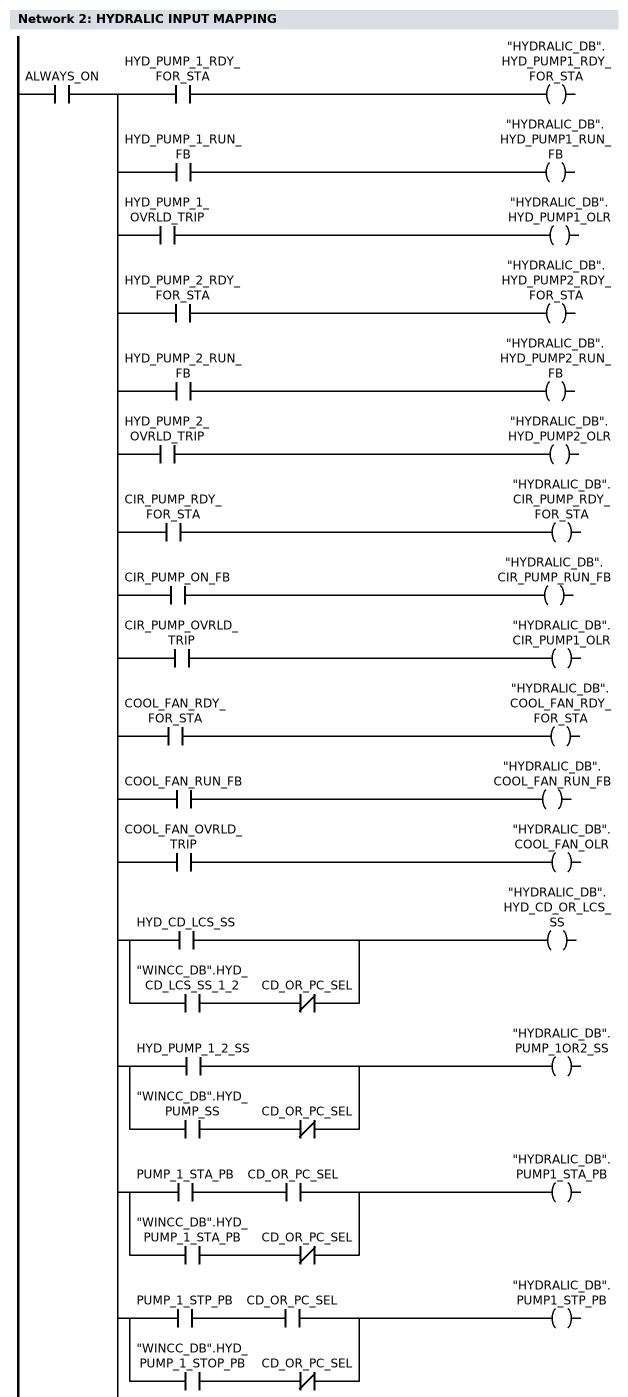
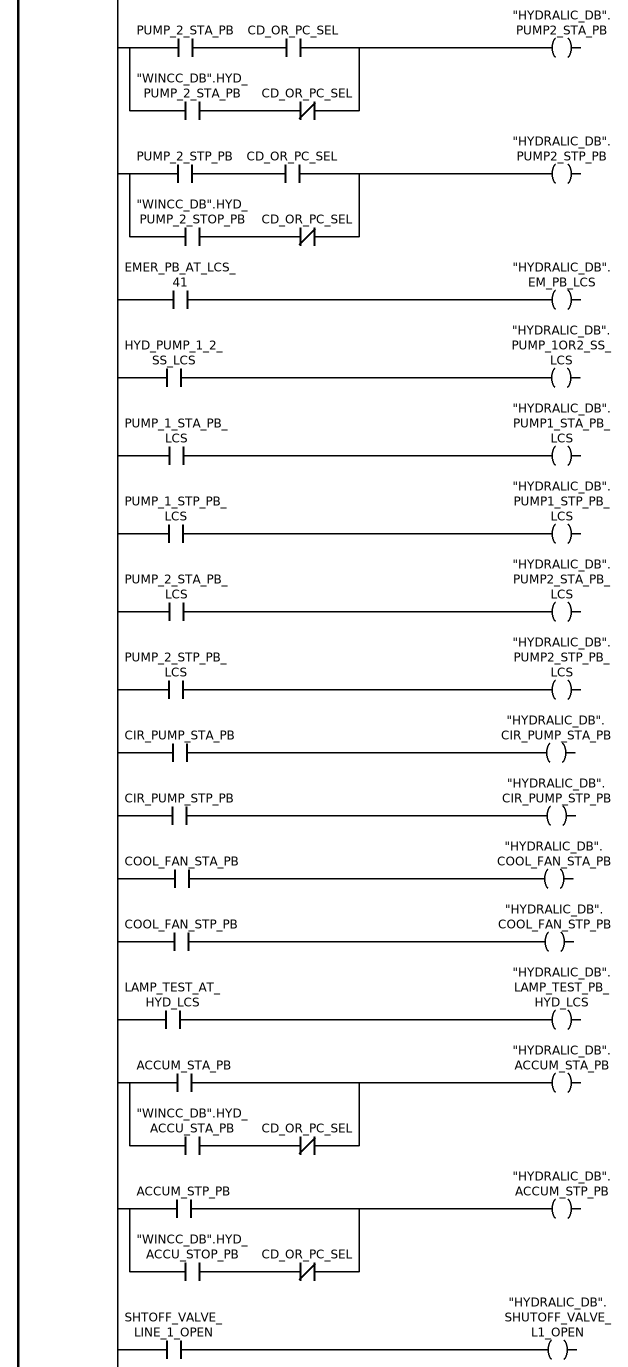
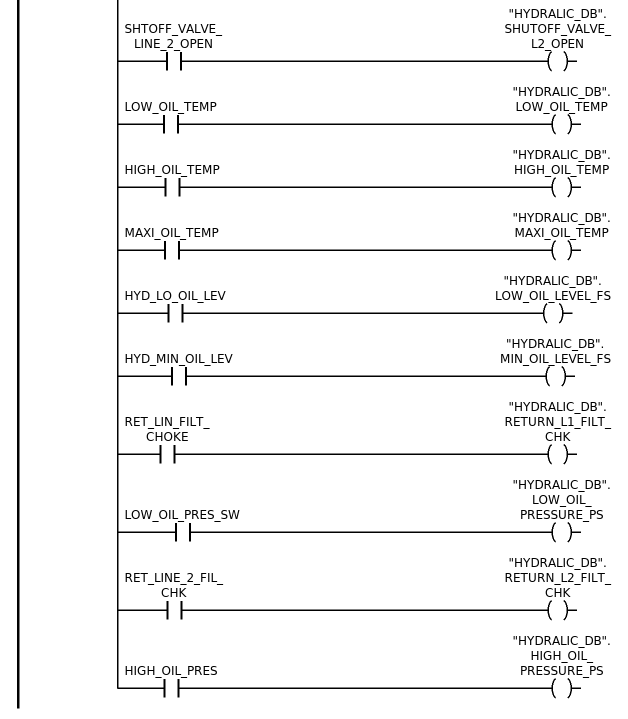
NETWORK
TITLE = HYDRALIC INPUT MAPPING
      A     "ALWAYS_ON";
      =     L 0.0;
      A     L 0.0;
      A     "HYD_PUMP_1_RDY_FOR_STA";
      =     "HYDRALIC_DB".HYD_PUMP1_RDY_FOR_STA;
      A     L 0.0;
      A     "HYD_PUMP_1_RUN_FB";
      =     "HYDRALIC_DB".HYD_PUMP1_RUN_FB;
      A     L 0.0;
      A     "HYD_PUMP_1_OVRLD_TRIP";
      =     "HYDRALIC_DB".HYD_PUMP1_OLR;
      A     L 0.0;
      A     "HYD_PUMP_2_RDY_FOR_STA";
      =     "HYDRALIC_DB".HYD_PUMP2_RDY_FOR_STA;
      A     L 0.0;
      A     "HYD_PUMP_2_RUN_FB";
      =     "HYDRALIC_DB".HYD_PUMP2_RUN_FB;
      A     L 0.0;
      A     "HYD_PUMP_2_OVRLD_TRIP";
      =     "HYDRALIC_DB".HYD_PUMP2_OLR;
      A     L 0.0;
      A     "CIR_PUMP_RDY_FOR_STA";
      =     "HYDRALIC_DB".CIR_PUMP_RDY_FOR_STA;
      A     L 0.0;
      A     "CIR_PUMP_ON_FB";
      =     "HYDRALIC_DB".CIR_PUMP_RUN_FB;
      A     L 0.0;
      A     "CIR_PUMP_OVRLD_TRIP";
      =     "HYDRALIC_DB".CIR_PUMP1_OLR;
      A     L 0.0;
      A     "COOL_FAN_RDY_FOR_STA";
      =     "HYDRALIC_DB".COOL_FAN_RDY_FOR_STA;
      A     L 0.0;
      A     "COOL_FAN_RUN_FB";
      =     "HYDRALIC_DB".COOL_FAN_RUN_FB;
      A     L 0.0;
      A     "COOL_FAN_OVRLD_TRIP";
      =     "HYDRALIC_DB".COOL_FAN_OLR;
      A     L 0.0;
      A(;
      O     "HYD_CD_LCS_SS";
      O;
      A     "WINCC_DB".HYD_CD_LCS_SS_1_2;
      AN    "CD_OR_PC_SEL";
      );
      =     "HYDRALIC_DB".HYD_CD_OR_LCS_SS;
      A     L 0.0;
      A(;
      O     "HYD_PUMP_1_2_SS";
      O;
      A     "WINCC_DB".HYD_PUMP_SS;
      AN    "CD_OR_PC_SEL";
      );
      =     "HYDRALIC_DB".PUMP_1OR2_SS;
      A     L 0.0;
      A(;
      A     "PUMP_1_STA_PB";
      A     "CD_OR_PC_SEL";
      O;
      A     "WINCC_DB".HYD_PUMP_1_STA_PB;
      AN    "CD_OR_PC_SEL";
      );
      =     "HYDRALIC_DB".PUMP1_STA_PB;
      A     L 0.0;
      A(;
      A     "PUMP_1_STP_PB";
      A     "CD_OR_PC_SEL";
      O;
      A     "WINCC_DB".HYD_PUMP_1_STOP_PB;
      AN    "CD_OR_PC_SEL";
      );
      =     "HYDRALIC_DB".PUMP1_STP_PB;
      A     L 0.0;
      A(;
      A     "PUMP_2_STA_PB";
      A     "CD_OR_PC_SEL";
      O;
      A     "WINCC_DB".HYD_PUMP_2_STA_PB;
      AN    "CD_OR_PC_SEL";
      );
      =     "HYDRALIC_DB".PUMP2_STA_PB;
      A     L 0.0;
      A(;
      A     "PUMP_2_STP_PB";
      A     "CD_OR_PC_SEL";
      O;
      A     "WINCC_DB".HYD_PUMP_2_STOP_PB;
      AN    "CD_OR_PC_SEL";
      );
      =     "HYDRALIC_DB".PUMP2_STP_PB;
      A     L 0.0;
      A     "EMER_PB_AT_LCS_41";
      =     "HYDRALIC_DB".EM_PB_LCS;
      A     L 0.0;
      A     "HYD_PUMP_1_2_SS_LCS";
      =     "HYDRALIC_DB".PUMP_1OR2_SS_LCS;
      A     L 0.0;
      A     "PUMP_1_STA_PB_LCS";
      =     "HYDRALIC_DB".PUMP1_STA_PB_LCS;
      A     L 0.0;
      A     "PUMP_1_STP_PB_LCS";
      =     "HYDRALIC_DB".PUMP1_STP_PB_LCS;
      A     L 0.0;
      A     "PUMP_2_STA_PB_LCS";
      =     "HYDRALIC_DB".PUMP2_STA_PB_LCS;
      A     L 0.0;
      A     "PUMP_2_STP_PB_LCS";
      =     "HYDRALIC_DB".PUMP2_STP_PB_LCS;
      A     L 0.0;
      A     "CIR_PUMP_STA_PB";
      =     "HYDRALIC_DB".CIR_PUMP_STA_PB;
      A     L 0.0;
      A     "CIR_PUMP_STP_PB";
      =     "HYDRALIC_DB".CIR_PUMP_STP_PB;
      A     L 0.0;
      A     "COOL_FAN_STA_PB";
      =     "HYDRALIC_DB".COOL_FAN_STA_PB;
      A     L 0.0;
      A     "COOL_FAN_STP_PB";
      =     "HYDRALIC_DB".COOL_FAN_STP_PB;
      A     L 0.0;
      A     "LAMP_TEST_AT_HYD_LCS";
      =     "HYDRALIC_DB".LAMP_TEST_PB_HYD_LCS;
      A     L 0.0;
      A(;
      O     "ACCUM_STA_PB";
      O;
      A     "WINCC_DB".HYD_ACCU_STA_PB;
      AN    "CD_OR_PC_SEL";
      );
      =     "HYDRALIC_DB".ACCUM_STA_PB;
      A     L 0.0;
      A(;
      O     "ACCUM_STP_PB";
      O;
      A     "WINCC_DB".HYD_ACCU_STOP_PB;
      AN    "CD_OR_PC_SEL";
      );
      =     "HYDRALIC_DB".ACCUM_STP_PB;
      A     L 0.0;
      A     "SHTOFF_VALVE_LINE_1_OPEN";
      =     "HYDRALIC_DB".SHUTOFF_VALVE_L1_OPEN;
      A     L 0.0;
      A     "SHTOFF_VALVE_LINE_2_OPEN";
      =     "HYDRALIC_DB".SHUTOFF_VALVE_L2_OPEN;
      A     L 0.0;
      A     "LOW_OIL_TEMP";
      =     "HYDRALIC_DB".LOW_OIL_TEMP;
      A     L 0.0;
      A     "HIGH_OIL_TEMP";
      =     "HYDRALIC_DB".HIGH_OIL_TEMP;
      A     L 0.0;
      A     "MAXI_OIL_TEMP";
      =     "HYDRALIC_DB".MAXI_OIL_TEMP;
      A     L 0.0;
      A     "HYD_LO_OIL_LEV";
      =     "HYDRALIC_DB".LOW_OIL_LEVEL_FS;
      A     L 0.0;
      A     "HYD_MIN_OIL_LEV";
      =     "HYDRALIC_DB".MIN_OIL_LEVEL_FS;
      A     L 0.0;
      A     "RET_LIN_FILT_CHOKE";
      =     "HYDRALIC_DB".RETURN_L1_FILT_CHK;
      A     L 0.0;
      A     "LOW_OIL_PRES_SW";
      =     "HYDRALIC_DB".LOW_OIL_PRESSURE_PS;
      A     L 0.0;
      A     "RET_LINE_2_FIL_CHK";
      =     "HYDRALIC_DB".RETURN_L2_FILT_CHK;
      A     L 0.0;
      A     "HIGH_OIL_PRES";
      =     "HYDRALIC_DB".HIGH_OIL_PRESSURE_PS;
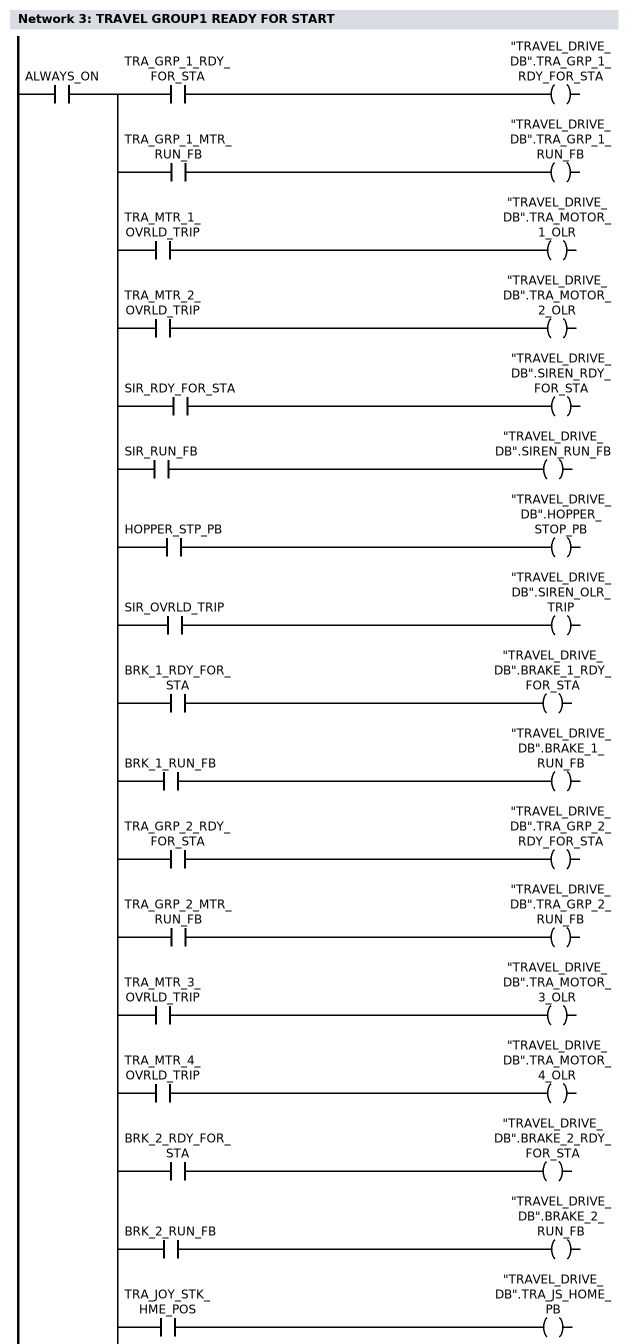
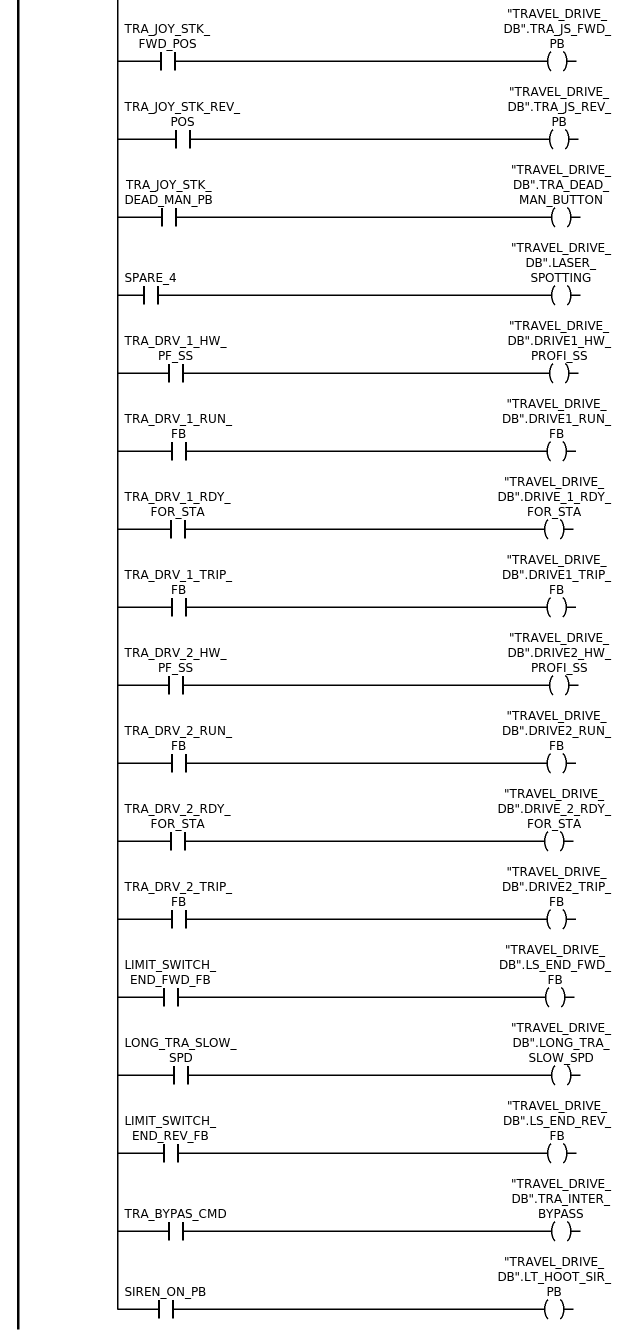
NETWORK
TITLE = TRAVEL GROUP1 READY FOR START
      A     "ALWAYS_ON";
      =     L 0.0;
      A     L 0.0;
      A     "TRA_GRP_1_RDY_FOR_STA";
      =     "TRAVEL_DRIVE_DB".TRA_GRP_1_RDY_FOR_STA;
      A     L 0.0;
      A     "TRA_GRP_1_MTR_RUN_FB";
      =     "TRAVEL_DRIVE_DB".TRA_GRP_1_RUN_FB;
      A     L 0.0;
      A     "TRA_MTR_1_OVRLD_TRIP";
      =     "TRAVEL_DRIVE_DB".TRA_MOTOR_1_OLR;
      A     L 0.0;
      A     "TRA_MTR_2_OVRLD_TRIP";
      =     "TRAVEL_DRIVE_DB".TRA_MOTOR_2_OLR;
      A     L 0.0;
      A     "SIR_RDY_FOR_STA";
      =     "TRAVEL_DRIVE_DB".SIREN_RDY_FOR_STA;
      A     L 0.0;
      A     "SIR_RUN_FB";
      =     "TRAVEL_DRIVE_DB".SIREN_RUN_FB;
      A     L 0.0;
      A     "HOPPER_STP_PB";
      =     "TRAVEL_DRIVE_DB".HOPPER_STOP_PB;
      A     L 0.0;
      A     "SIR_OVRLD_TRIP";
      =     "TRAVEL_DRIVE_DB".SIREN_OLR_TRIP;
      A     L 0.0;
      A     "BRK_1_RDY_FOR_STA";
      =     "TRAVEL_DRIVE_DB".BRAKE_1_RDY_FOR_STA;
      A     L 0.0;
      A     "BRK_1_RUN_FB";
      =     "TRAVEL_DRIVE_DB".BRAKE_1_RUN_FB;
      A     L 0.0;
      A     "TRA_GRP_2_RDY_FOR_STA";
      =     "TRAVEL_DRIVE_DB".TRA_GRP_2_RDY_FOR_STA;
      A     L 0.0;
      A     "TRA_GRP_2_MTR_RUN_FB";
      =     "TRAVEL_DRIVE_DB".TRA_GRP_2_RUN_FB;
      A     L 0.0;
      A     "TRA_MTR_3_OVRLD_TRIP";
      =     "TRAVEL_DRIVE_DB".TRA_MOTOR_3_OLR;
      A     L 0.0;
      A     "TRA_MTR_4_OVRLD_TRIP";
      =     "TRAVEL_DRIVE_DB".TRA_MOTOR_4_OLR;
      A     L 0.0;
      A     "BRK_2_RDY_FOR_STA";
      =     "TRAVEL_DRIVE_DB".BRAKE_2_RDY_FOR_STA;
      A     L 0.0;
      A     "BRK_2_RUN_FB";
      =     "TRAVEL_DRIVE_DB".BRAKE_2_RUN_FB;
      A     L 0.0;
      A     "TRA_JOY_STK_HME_POS";
      =     "TRAVEL_DRIVE_DB".TRA_JS_HOME_PB;
      A     L 0.0;
      A     "TRA_JOY_STK_FWD_POS";
      =     "TRAVEL_DRIVE_DB".TRA_JS_FWD_PB;
      A     L 0.0;
      A     "TRA_JOY_STK_REV_POS";
      =     "TRAVEL_DRIVE_DB".TRA_JS_REV_PB;
      A     L 0.0;
      A     "TRA_JOY_STK_DEAD_MAN_PB";
      =     "TRAVEL_DRIVE_DB".TRA_DEAD_MAN_BUTTON;
      A     L 0.0;
      A     "SPARE_4";
      =     "TRAVEL_DRIVE_DB".LASER_SPOTTING;
      A     L 0.0;
      A     "TRA_DRV_1_HW_PF_SS";
      =     "TRAVEL_DRIVE_DB".DRIVE1_HW_PROFI_SS;
      A     L 0.0;
      A     "TRA_DRV_1_RUN_FB";
      =     "TRAVEL_DRIVE_DB".DRIVE1_RUN_FB;
      A     L 0.0;
      A     "TRA_DRV_1_RDY_FOR_STA";
      =     "TRAVEL_DRIVE_DB".DRIVE_1_RDY_FOR_STA;
      A     L 0.0;
      A     "TRA_DRV_1_TRIP_FB";
      =     "TRAVEL_DRIVE_DB".DRIVE1_TRIP_FB;
      A     L 0.0;
      A     "TRA_DRV_2_HW_PF_SS";
      =     "TRAVEL_DRIVE_DB".DRIVE2_HW_PROFI_SS;
      A     L 0.0;
      A     "TRA_DRV_2_RUN_FB";
      =     "TRAVEL_DRIVE_DB".DRIVE2_RUN_FB;
      A     L 0.0;
      A     "TRA_DRV_2_RDY_FOR_STA";
      =     "TRAVEL_DRIVE_DB".DRIVE_2_RDY_FOR_STA;
      A     L 0.0;
      A     "TRA_DRV_2_TRIP_FB";
      =     "TRAVEL_DRIVE_DB".DRIVE2_TRIP_FB;
      A     L 0.0;
      A     "LIMIT_SWITCH_END_FWD_FB";
      =     "TRAVEL_DRIVE_DB".LS_END_FWD_FB;
      A     L 0.0;
      A     "LONG_TRA_SLOW_SPD";
      =     "TRAVEL_DRIVE_DB".LONG_TRA_SLOW_SPD;
      A     L 0.0;
      A     "LIMIT_SWITCH_END_REV_FB";
      =     "TRAVEL_DRIVE_DB".LS_END_REV_FB;
      A     L 0.0;
      A     "TRA_BYPAS_CMD";
      =     "TRAVEL_DRIVE_DB".TRA_INTER_BYPASS;
      A     L 0.0;
      A     "SIREN_ON_PB";
      =     "TRAVEL_DRIVE_DB".LT_HOOT_SIR_PB;
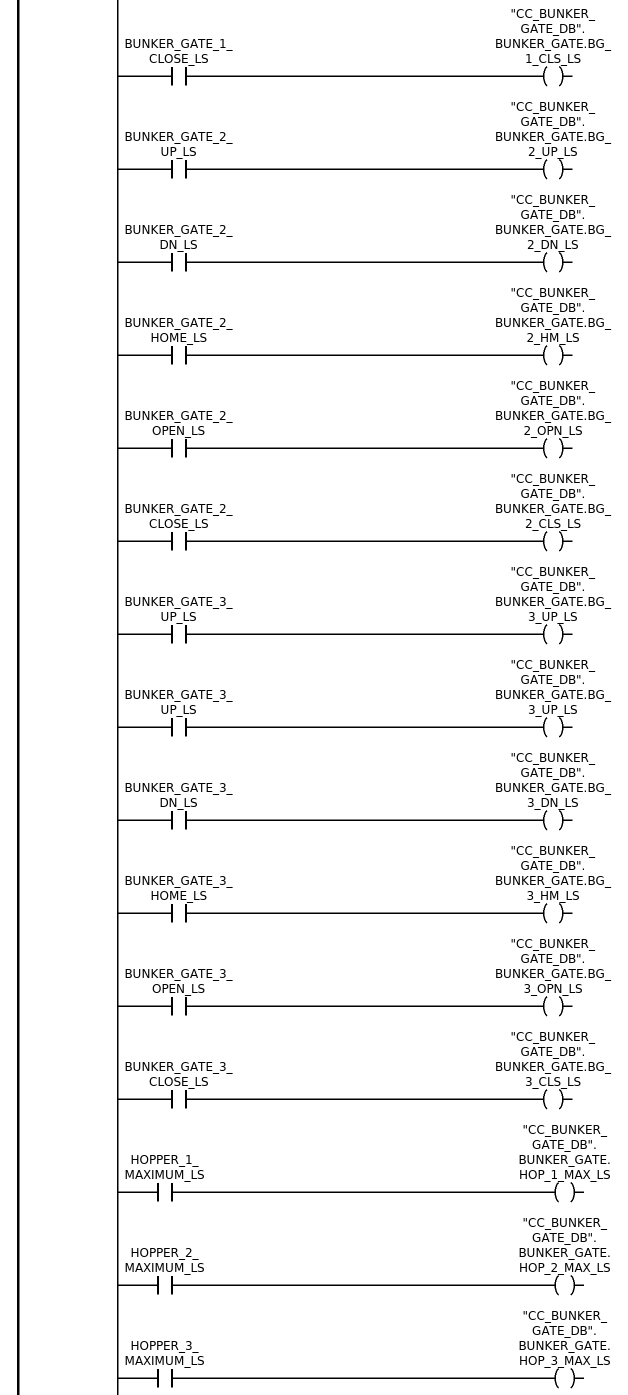
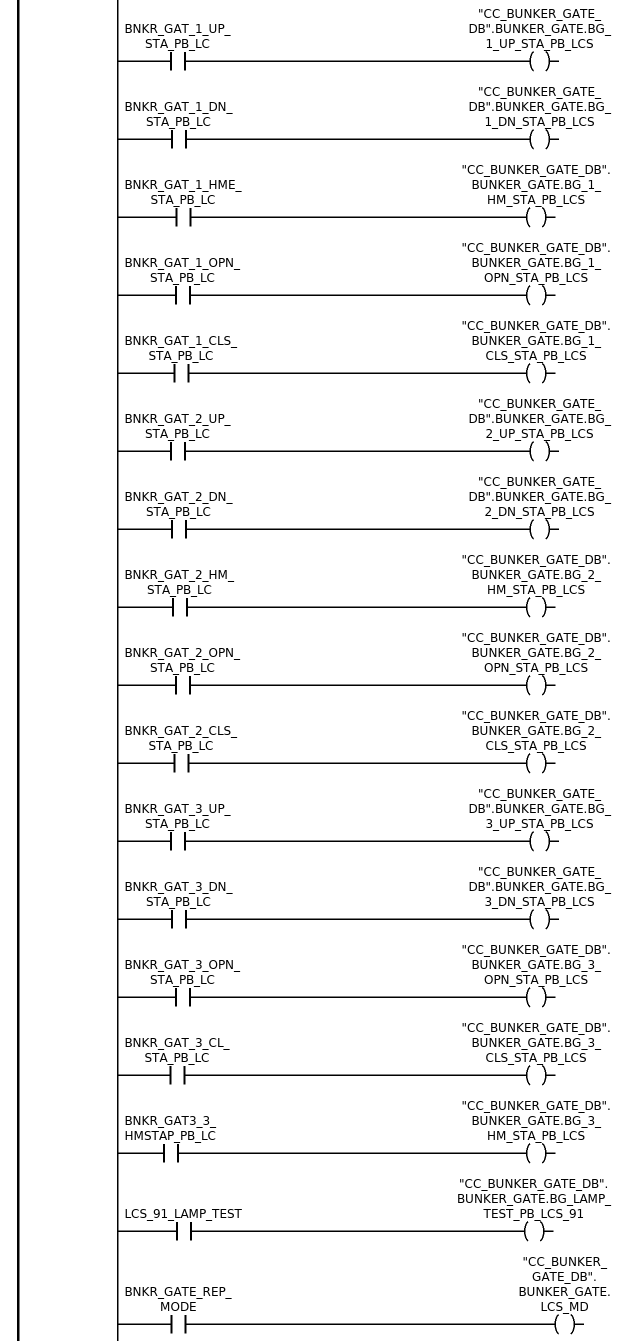
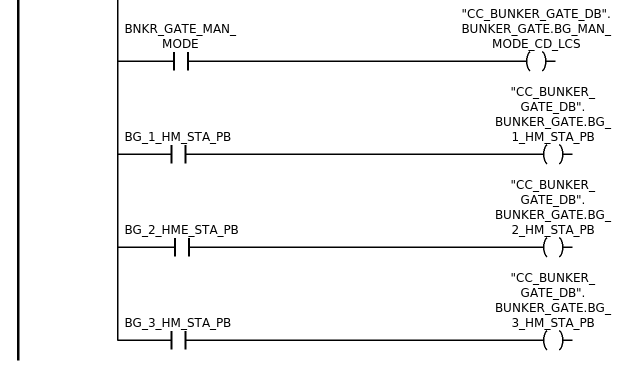
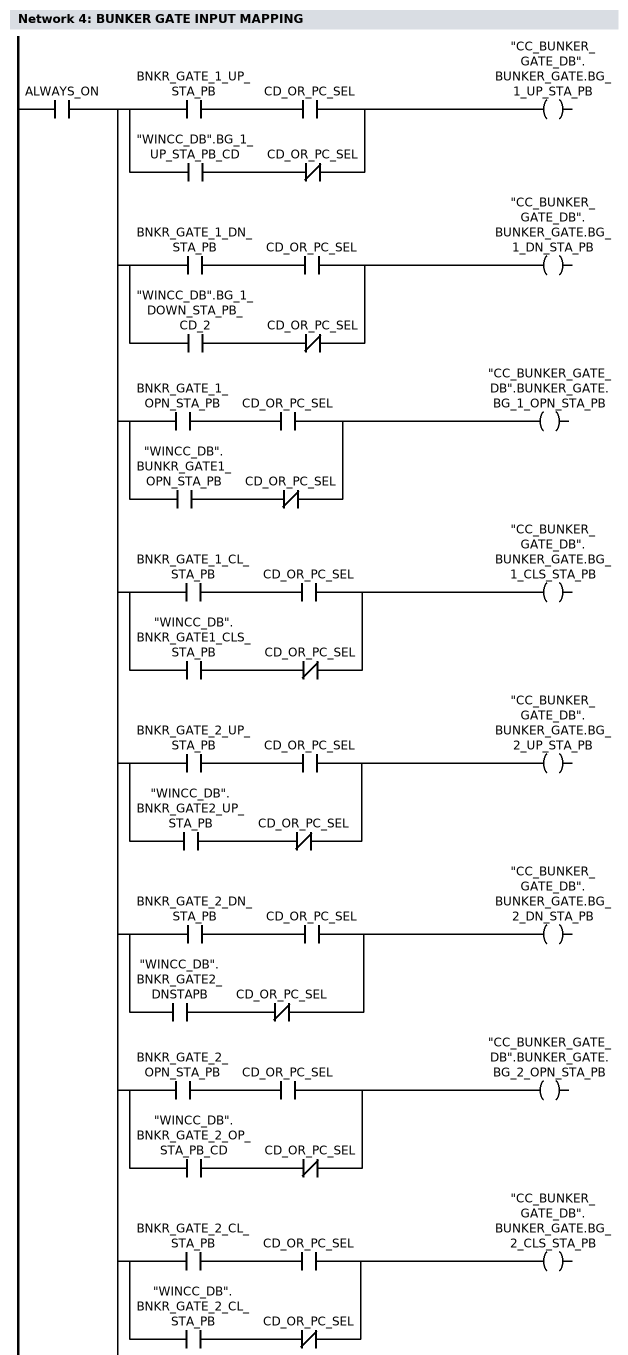
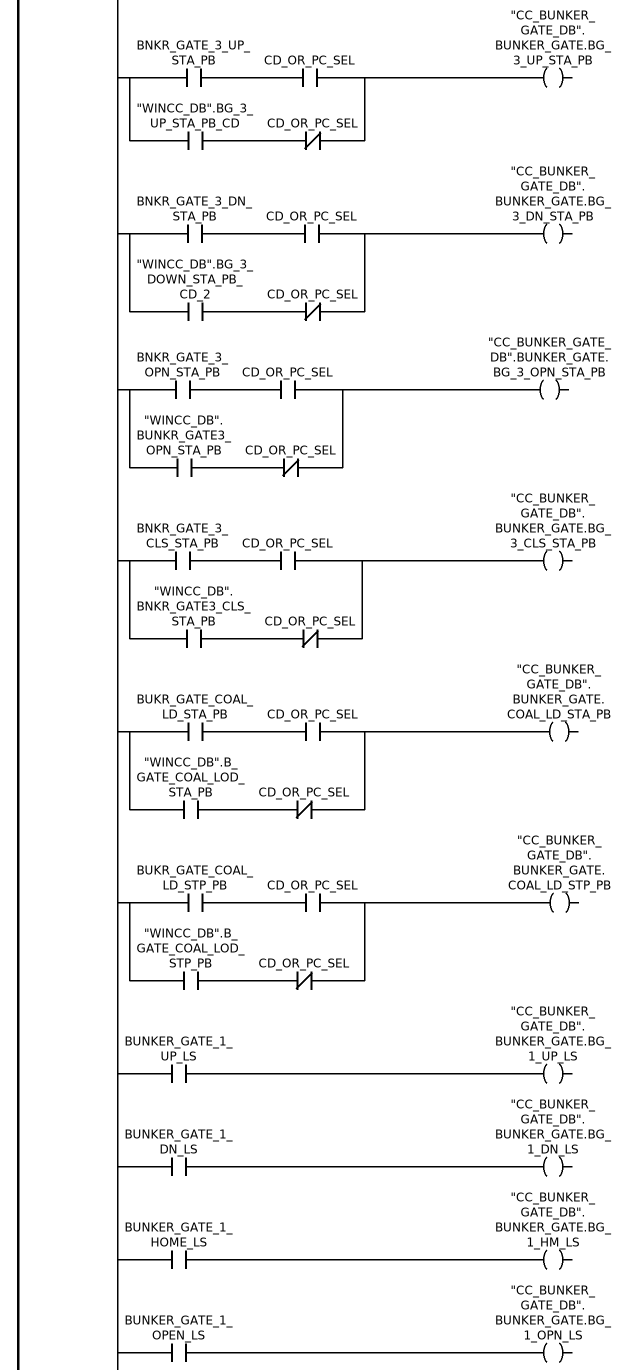
NETWORK
TITLE = BUNKER GATE INPUT MAPPING
      A     "ALWAYS_ON";
      =     L 0.0;
      A     L 0.0;
      A(;
      A     "BNKR_GATE_1_UP_STA_PB";
      A     "CD_OR_PC_SEL";
      O;
      A     "WINCC_DB".BG_1_UP_STA_PB_CD;
      AN    "CD_OR_PC_SEL";
      );
      =     "CC_BUNKER_GATE_DB".BUNKER_GATE.BG_1_UP_STA_PB;
      A     L 0.0;
      A(;
      A     "BNKR_GATE_1_DN_STA_PB";
      A     "CD_OR_PC_SEL";
      O;
      A     "WINCC_DB".BG_1_DOWN_STA_PB_CD_2;
      AN    "CD_OR_PC_SEL";
      );
      =     "CC_BUNKER_GATE_DB".BUNKER_GATE.BG_1_DN_STA_PB;
      A     L 0.0;
      A(;
      A     "BNKR_GATE_1_OPN_STA_PB";
      A     "CD_OR_PC_SEL";
      O;
      A     "WINCC_DB".BUNKR_GATE1_OPN_STA_PB;
      AN    "CD_OR_PC_SEL";
      );
      =     "CC_BUNKER_GATE_DB".BUNKER_GATE.BG_1_OPN_STA_PB;
      A     L 0.0;
      A(;
      A     "BNKR_GATE_1_CL_STA_PB";
      A     "CD_OR_PC_SEL";
      O;
      A     "WINCC_DB".BNKR_GATE1_CLS_STA_PB;
      AN    "CD_OR_PC_SEL";
      );
      =     "CC_BUNKER_GATE_DB".BUNKER_GATE.BG_1_CLS_STA_PB;
      A     L 0.0;
      A(;
      A     "BNKR_GATE_2_UP_STA_PB";
      A     "CD_OR_PC_SEL";
      O;
      A     "WINCC_DB".BNKR_GATE2_UP_STA_PB;
      AN    "CD_OR_PC_SEL";
      );
      =     "CC_BUNKER_GATE_DB".BUNKER_GATE.BG_2_UP_STA_PB;
      A     L 0.0;
      A(;
      A     "BNKR_GATE_2_DN_STA_PB";
      A     "CD_OR_PC_SEL";
      O;
      A     "WINCC_DB".BNKR_GATE2_DNSTAPB;
      AN    "CD_OR_PC_SEL";
      );
      =     "CC_BUNKER_GATE_DB".BUNKER_GATE.BG_2_DN_STA_PB;
      A     L 0.0;
      A(;
      A     "BNKR_GATE_2_OPN_STA_PB";
      A     "CD_OR_PC_SEL";
      O;
      A     "WINCC_DB".BNKR_GATE_2_OP_STA_PB_CD;
      AN    "CD_OR_PC_SEL";
      );
      =     "CC_BUNKER_GATE_DB".BUNKER_GATE.BG_2_OPN_STA_PB;
      A     L 0.0;
      A(;
      A     "BNKR_GATE_2_CL_STA_PB";
      A     "CD_OR_PC_SEL";
      O;
      A     "WINCC_DB".BNKR_GATE_2_CL_STA_PB;
      AN    "CD_OR_PC_SEL";
      );
      =     "CC_BUNKER_GATE_DB".BUNKER_GATE.BG_2_CLS_STA_PB;
      A     L 0.0;
      A(;
      A     "BNKR_GATE_3_UP_STA_PB";
      A     "CD_OR_PC_SEL";
      O;
      A     "WINCC_DB".BG_3_UP_STA_PB_CD;
      AN    "CD_OR_PC_SEL";
      );
      =     "CC_BUNKER_GATE_DB".BUNKER_GATE.BG_3_UP_STA_PB;
      A     L 0.0;
      A(;
      A     "BNKR_GATE_3_DN_STA_PB";
      A     "CD_OR_PC_SEL";
      O;
      A     "WINCC_DB".BG_3_DOWN_STA_PB_CD_2;
      AN    "CD_OR_PC_SEL";
      );
      =     "CC_BUNKER_GATE_DB".BUNKER_GATE.BG_3_DN_STA_PB;
      A     L 0.0;
      A(;
      A     "BNKR_GATE_3_OPN_STA_PB";
      A     "CD_OR_PC_SEL";
      O;
      A     "WINCC_DB".BUNKR_GATE3_OPN_STA_PB;
      AN    "CD_OR_PC_SEL";
      );
      =     "CC_BUNKER_GATE_DB".BUNKER_GATE.BG_3_OPN_STA_PB;
      A     L 0.0;
      A(;
      A     "BNKR_GATE_3_CLS_STA_PB";
      A     "CD_OR_PC_SEL";
      O;
      A     "WINCC_DB".BNKR_GATE3_CLS_STA_PB;
      AN    "CD_OR_PC_SEL";
      );
      =     "CC_BUNKER_GATE_DB".BUNKER_GATE.BG_3_CLS_STA_PB;
      A     L 0.0;
      A(;
      A     "BUKR_GATE_COAL_LD_STA_PB";
      A     "CD_OR_PC_SEL";
      O;
      A     "WINCC_DB".B_GATE_COAL_LOD_STA_PB;
      AN    "CD_OR_PC_SEL";
      );
      =     "CC_BUNKER_GATE_DB".BUNKER_GATE.COAL_LD_STA_PB;
      A     L 0.0;
      A(;
      A     "BUKR_GATE_COAL_LD_STP_PB";
      A     "CD_OR_PC_SEL";
      O;
      A     "WINCC_DB".B_GATE_COAL_LOD_STP_PB;
      AN    "CD_OR_PC_SEL";
      );
      =     "CC_BUNKER_GATE_DB".BUNKER_GATE.COAL_LD_STP_PB;
      A     L 0.0;
      A     "BUNKER_GATE_1_UP_LS";
      =     "CC_BUNKER_GATE_DB".BUNKER_GATE.BG_1_UP_LS;
      A     L 0.0;
      A     "BUNKER_GATE_1_DN_LS";
      =     "CC_BUNKER_GATE_DB".BUNKER_GATE.BG_1_DN_LS;
      A     L 0.0;
      A     "BUNKER_GATE_1_HOME_LS";
      =     "CC_BUNKER_GATE_DB".BUNKER_GATE.BG_1_HM_LS;
      A     L 0.0;
      A     "BUNKER_GATE_1_OPEN_LS";
      =     "CC_BUNKER_GATE_DB".BUNKER_GATE.BG_1_OPN_LS;
      A     L 0.0;
      A     "BUNKER_GATE_1_CLOSE_LS";
      =     "CC_BUNKER_GATE_DB".BUNKER_GATE.BG_1_CLS_LS;
      A     L 0.0;
      A     "BUNKER_GATE_2_UP_LS";
      =     "CC_BUNKER_GATE_DB".BUNKER_GATE.BG_2_UP_LS;
      A     L 0.0;
      A     "BUNKER_GATE_2_DN_LS";
      =     "CC_BUNKER_GATE_DB".BUNKER_GATE.BG_2_DN_LS;
      A     L 0.0;
      A     "BUNKER_GATE_2_HOME_LS";
      =     "CC_BUNKER_GATE_DB".BUNKER_GATE.BG_2_HM_LS;
      A     L 0.0;
      A     "BUNKER_GATE_2_OPEN_LS";
      =     "CC_BUNKER_GATE_DB".BUNKER_GATE.BG_2_OPN_LS;
      A     L 0.0;
      A     "BUNKER_GATE_2_CLOSE_LS";
      =     "CC_BUNKER_GATE_DB".BUNKER_GATE.BG_2_CLS_LS;
      A     L 0.0;
      A     "BUNKER_GATE_3_UP_LS";
      =     "CC_BUNKER_GATE_DB".BUNKER_GATE.BG_3_UP_LS;
      A     L 0.0;
      A     "BUNKER_GATE_3_UP_LS";
      =     "CC_BUNKER_GATE_DB".BUNKER_GATE.BG_3_UP_LS;
      A     L 0.0;
      A     "BUNKER_GATE_3_DN_LS";
      =     "CC_BUNKER_GATE_DB".BUNKER_GATE.BG_3_DN_LS;
      A     L 0.0;
      A     "BUNKER_GATE_3_HOME_LS";
      =     "CC_BUNKER_GATE_DB".BUNKER_GATE.BG_3_HM_LS;
      A     L 0.0;
      A     "BUNKER_GATE_3_OPEN_LS";
      =     "CC_BUNKER_GATE_DB".BUNKER_GATE.BG_3_OPN_LS;
      A     L 0.0;
      A     "BUNKER_GATE_3_CLOSE_LS";
      =     "CC_BUNKER_GATE_DB".BUNKER_GATE.BG_3_CLS_LS;
      A     L 0.0;
      A     "HOPPER_1_MAXIMUM_LS";
      =     "CC_BUNKER_GATE_DB".BUNKER_GATE.HOP_1_MAX_LS;
      A     L 0.0;
      A     "HOPPER_2_MAXIMUM_LS";
      =     "CC_BUNKER_GATE_DB".BUNKER_GATE.HOP_2_MAX_LS;
      A     L 0.0;
      A     "HOPPER_3_MAXIMUM_LS";
      =     "CC_BUNKER_GATE_DB".BUNKER_GATE.HOP_3_MAX_LS;
      A     L 0.0;
      A     "BNKR_GAT_1_UP_STA_PB_LC";
      =     "CC_BUNKER_GATE_DB".BUNKER_GATE.BG_1_UP_STA_PB_LCS;
      A     L 0.0;
      A     "BNKR_GAT_1_DN_STA_PB_LC";
      =     "CC_BUNKER_GATE_DB".BUNKER_GATE.BG_1_DN_STA_PB_LCS;
      A     L 0.0;
      A     "BNKR_GAT_1_HME_STA_PB_LC";
      =     "CC_BUNKER_GATE_DB".BUNKER_GATE.BG_1_HM_STA_PB_LCS;
      A     L 0.0;
      A     "BNKR_GAT_1_OPN_STA_PB_LC";
      =     "CC_BUNKER_GATE_DB".BUNKER_GATE.BG_1_OPN_STA_PB_LCS;
      A     L 0.0;
      A     "BNKR_GAT_1_CLS_STA_PB_LC";
      =     "CC_BUNKER_GATE_DB".BUNKER_GATE.BG_1_CLS_STA_PB_LCS;
      A     L 0.0;
      A     "BNKR_GAT_2_UP_STA_PB_LC";
      =     "CC_BUNKER_GATE_DB".BUNKER_GATE.BG_2_UP_STA_PB_LCS;
      A     L 0.0;
      A     "BNKR_GAT_2_DN_STA_PB_LC";
      =     "CC_BUNKER_GATE_DB".BUNKER_GATE.BG_2_DN_STA_PB_LCS;
      A     L 0.0;
      A     "BNKR_GAT_2_HM_STA_PB_LC";
      =     "CC_BUNKER_GATE_DB".BUNKER_GATE.BG_2_HM_STA_PB_LCS;
      A     L 0.0;
      A     "BNKR_GAT_2_OPN_STA_PB_LC";
      =     "CC_BUNKER_GATE_DB".BUNKER_GATE.BG_2_OPN_STA_PB_LCS;
      A     L 0.0;
      A     "BNKR_GAT_2_CLS_STA_PB_LC";
      =     "CC_BUNKER_GATE_DB".BUNKER_GATE.BG_2_CLS_STA_PB_LCS;
      A     L 0.0;
      A     "BNKR_GAT_3_UP_STA_PB_LC";
      =     "CC_BUNKER_GATE_DB".BUNKER_GATE.BG_3_UP_STA_PB_LCS;
      A     L 0.0;
      A     "BNKR_GAT_3_DN_STA_PB_LC";
      =     "CC_BUNKER_GATE_DB".BUNKER_GATE.BG_3_DN_STA_PB_LCS;
      A     L 0.0;
      A     "BNKR_GAT_3_OPN_STA_PB_LC";
      =     "CC_BUNKER_GATE_DB".BUNKER_GATE.BG_3_OPN_STA_PB_LCS;
      A     L 0.0;
      A     "BNKR_GAT_3_CL_STA_PB_LC";
      =     "CC_BUNKER_GATE_DB".BUNKER_GATE.BG_3_CLS_STA_PB_LCS;
      A     L 0.0;
      A     "BNKR_GAT3_3_HMSTAP_PB_LC";
      =     "CC_BUNKER_GATE_DB".BUNKER_GATE.BG_3_HM_STA_PB_LCS;
      A     L 0.0;
      A     "LCS_91_LAMP_TEST";
      =     "CC_BUNKER_GATE_DB".BUNKER_GATE.BG_LAMP_TEST_PB_LCS_91;
      A     L 0.0;
      A     "BNKR_GATE_REP_MODE";
      =     "CC_BUNKER_GATE_DB".BUNKER_GATE.LCS_MD;
      A     L 0.0;
      A     "BNKR_GATE_MAN_MODE";
      =     "CC_BUNKER_GATE_DB".BUNKER_GATE.BG_MAN_MODE_CD_LCS;
      A     L 0.0;
      A     "BG_1_HM_STA_PB";
      =     "CC_BUNKER_GATE_DB".BUNKER_GATE.BG_1_HM_STA_PB;
      A     L 0.0;
      A     "BG_2_HME_STA_PB";
      =     "CC_BUNKER_GATE_DB".BUNKER_GATE.BG_2_HM_STA_PB;
      A     L 0.0;
      A     "BG_3_HM_STA_PB";
      =     "CC_BUNKER_GATE_DB".BUNKER_GATE.BG_3_HM_STA_PB;
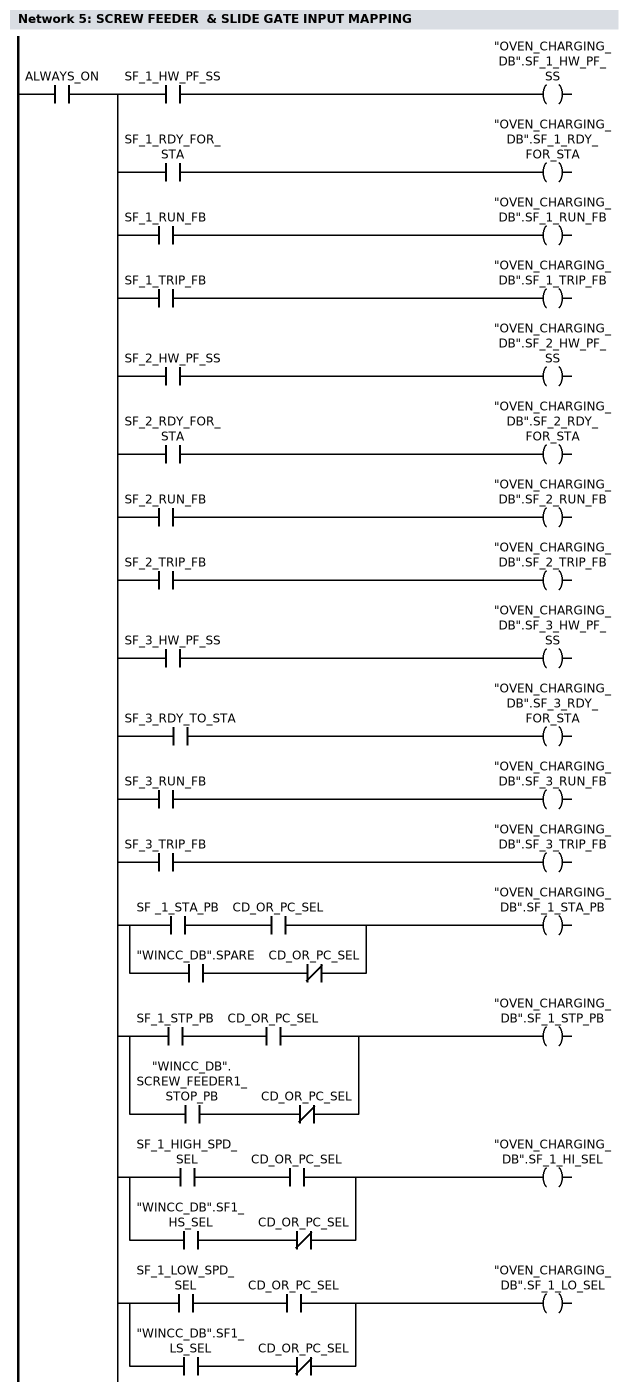
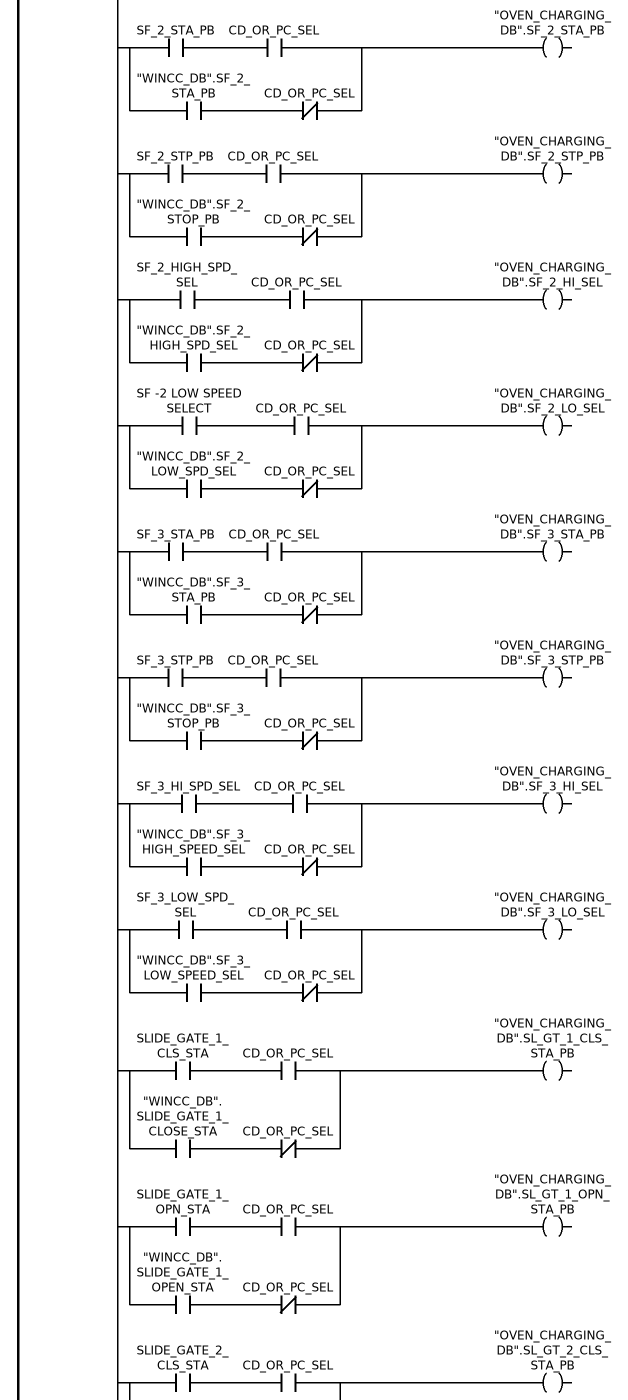
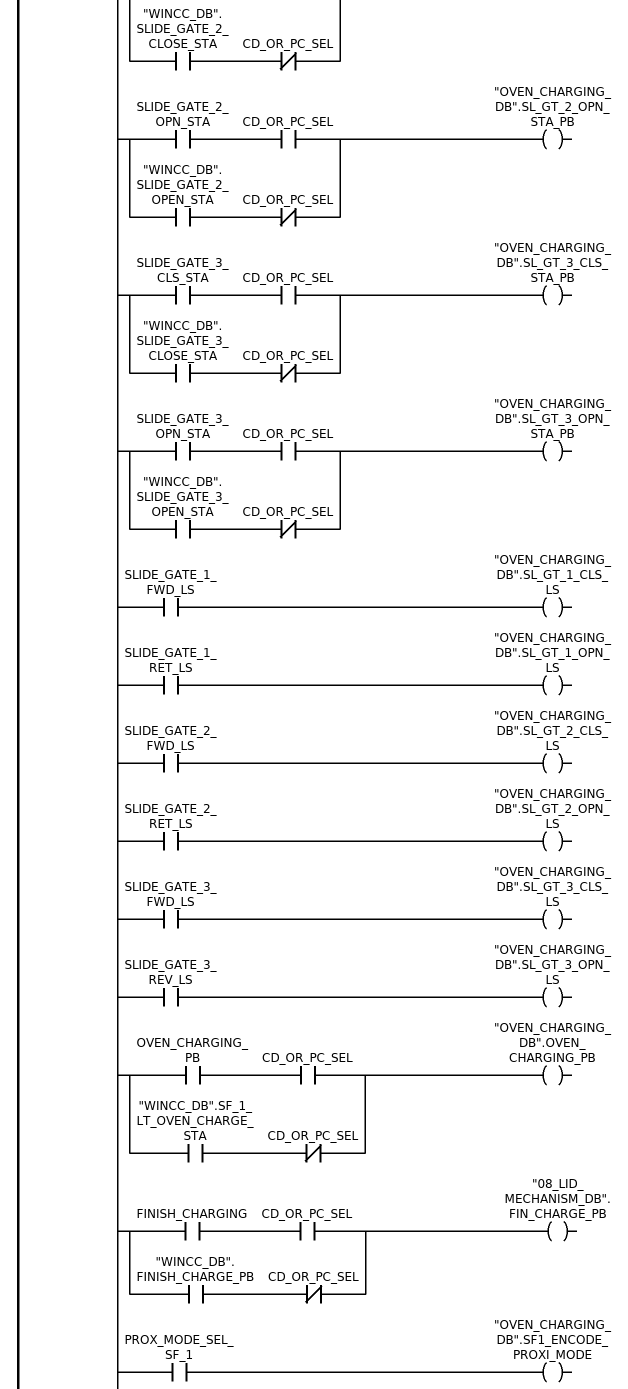
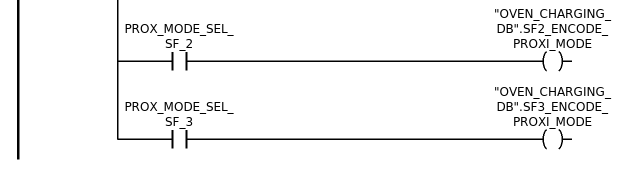
NETWORK
TITLE = SCREW FEEDER  & SLIDE GATE INPUT MAPPING
      A     "ALWAYS_ON";
      =     L 0.0;
      A     L 0.0;
      A     "SF_1_HW_PF_SS";
      =     "OVEN_CHARGING_DB".SF_1_HW_PF_SS;
      A     L 0.0;
      A     "SF_1_RDY_FOR_STA";
      =     "OVEN_CHARGING_DB".SF_1_RDY_FOR_STA;
      A     L 0.0;
      A     "SF_1_RUN_FB";
      =     "OVEN_CHARGING_DB".SF_1_RUN_FB;
      A     L 0.0;
      A     "SF_1_TRIP_FB";
      =     "OVEN_CHARGING_DB".SF_1_TRIP_FB;
      A     L 0.0;
      A     "SF_2_HW_PF_SS";
      =     "OVEN_CHARGING_DB".SF_2_HW_PF_SS;
      A     L 0.0;
      A     "SF_2_RDY_FOR_STA";
      =     "OVEN_CHARGING_DB".SF_2_RDY_FOR_STA;
      A     L 0.0;
      A     "SF_2_RUN_FB";
      =     "OVEN_CHARGING_DB".SF_2_RUN_FB;
      A     L 0.0;
      A     "SF_2_TRIP_FB";
      =     "OVEN_CHARGING_DB".SF_2_TRIP_FB;
      A     L 0.0;
      A     "SF_3_HW_PF_SS";
      =     "OVEN_CHARGING_DB".SF_3_HW_PF_SS;
      A     L 0.0;
      A     "SF_3_RDY_TO_STA";
      =     "OVEN_CHARGING_DB".SF_3_RDY_FOR_STA;
      A     L 0.0;
      A     "SF_3_RUN_FB";
      =     "OVEN_CHARGING_DB".SF_3_RUN_FB;
      A     L 0.0;
      A     "SF_3_TRIP_FB";
      =     "OVEN_CHARGING_DB".SF_3_TRIP_FB;
      A     L 0.0;
      A(;
      A     "SF _1_STA_PB";
      A     "CD_OR_PC_SEL";
      O;
      A     "WINCC_DB".SPARE;
      AN    "CD_OR_PC_SEL";
      );
      =     "OVEN_CHARGING_DB".SF_1_STA_PB;
      A     L 0.0;
      A(;
      A     "SF_1_STP_PB";
      A     "CD_OR_PC_SEL";
      O;
      A     "WINCC_DB".SCREW_FEEDER1_STOP_PB;
      AN    "CD_OR_PC_SEL";
      );
      =     "OVEN_CHARGING_DB".SF_1_STP_PB;
      A     L 0.0;
      A(;
      A     "SF_1_HIGH_SPD_SEL";
      A     "CD_OR_PC_SEL";
      O;
      A     "WINCC_DB".SF1_HS_SEL;
      AN    "CD_OR_PC_SEL";
      );
      =     "OVEN_CHARGING_DB".SF_1_HI_SEL;
      A     L 0.0;
      A(;
      A     "SF_1_LOW_SPD_SEL";
      A     "CD_OR_PC_SEL";
      O;
      A     "WINCC_DB".SF1_LS_SEL;
      AN    "CD_OR_PC_SEL";
      );
      =     "OVEN_CHARGING_DB".SF_1_LO_SEL;
      A     L 0.0;
      A(;
      A     "SF_2_STA_PB";
      A     "CD_OR_PC_SEL";
      O;
      A     "WINCC_DB".SF_2_STA_PB;
      AN    "CD_OR_PC_SEL";
      );
      =     "OVEN_CHARGING_DB".SF_2_STA_PB;
      A     L 0.0;
      A(;
      A     "SF_2_STP_PB";
      A     "CD_OR_PC_SEL";
      O;
      A     "WINCC_DB".SF_2_STOP_PB;
      AN    "CD_OR_PC_SEL";
      );
      =     "OVEN_CHARGING_DB".SF_2_STP_PB;
      A     L 0.0;
      A(;
      A     "SF_2_HIGH_SPD_SEL";
      A     "CD_OR_PC_SEL";
      O;
      A     "WINCC_DB".SF_2_HIGH_SPD_SEL;
      AN    "CD_OR_PC_SEL";
      );
      =     "OVEN_CHARGING_DB".SF_2_HI_SEL;
      A     L 0.0;
      A(;
      A     "SF -2 LOW SPEED SELECT";
      A     "CD_OR_PC_SEL";
      O;
      A     "WINCC_DB".SF_2_LOW_SPD_SEL;
      AN    "CD_OR_PC_SEL";
      );
      =     "OVEN_CHARGING_DB".SF_2_LO_SEL;
      A     L 0.0;
      A(;
      A     "SF_3_STA_PB";
      A     "CD_OR_PC_SEL";
      O;
      A     "WINCC_DB".SF_3_STA_PB;
      AN    "CD_OR_PC_SEL";
      );
      =     "OVEN_CHARGING_DB".SF_3_STA_PB;
      A     L 0.0;
      A(;
      A     "SF_3_STP_PB";
      A     "CD_OR_PC_SEL";
      O;
      A     "WINCC_DB".SF_3_STOP_PB;
      AN    "CD_OR_PC_SEL";
      );
      =     "OVEN_CHARGING_DB".SF_3_STP_PB;
      A     L 0.0;
      A(;
      A     "SF_3_HI_SPD_SEL";
      A     "CD_OR_PC_SEL";
      O;
      A     "WINCC_DB".SF_3_HIGH_SPEED_SEL;
      AN    "CD_OR_PC_SEL";
      );
      =     "OVEN_CHARGING_DB".SF_3_HI_SEL;
      A     L 0.0;
      A(;
      A     "SF_3_LOW_SPD_SEL";
      A     "CD_OR_PC_SEL";
      O;
      A     "WINCC_DB".SF_3_LOW_SPEED_SEL;
      AN    "CD_OR_PC_SEL";
      );
      =     "OVEN_CHARGING_DB".SF_3_LO_SEL;
      A     L 0.0;
      A(;
      A     "SLIDE_GATE_1_CLS_STA";
      A     "CD_OR_PC_SEL";
      O;
      A     "WINCC_DB".SLIDE_GATE_1_CLOSE_STA;
      AN    "CD_OR_PC_SEL";
      );
      =     "OVEN_CHARGING_DB".SL_GT_1_CLS_STA_PB;
      A     L 0.0;
      A(;
      A     "SLIDE_GATE_1_OPN_STA";
      A     "CD_OR_PC_SEL";
      O;
      A     "WINCC_DB".SLIDE_GATE_1_OPEN_STA;
      AN    "CD_OR_PC_SEL";
      );
      =     "OVEN_CHARGING_DB".SL_GT_1_OPN_STA_PB;
      A     L 0.0;
      A(;
      A     "SLIDE_GATE_2_CLS_STA";
      A     "CD_OR_PC_SEL";
      O;
      A     "WINCC_DB".SLIDE_GATE_2_CLOSE_STA;
      AN    "CD_OR_PC_SEL";
      );
      =     "OVEN_CHARGING_DB".SL_GT_2_CLS_STA_PB;
      A     L 0.0;
      A(;
      A     "SLIDE_GATE_2_OPN_STA";
      A     "CD_OR_PC_SEL";
      O;
      A     "WINCC_DB".SLIDE_GATE_2_OPEN_STA;
      AN    "CD_OR_PC_SEL";
      );
      =     "OVEN_CHARGING_DB".SL_GT_2_OPN_STA_PB;
      A     L 0.0;
      A(;
      A     "SLIDE_GATE_3_CLS_STA";
      A     "CD_OR_PC_SEL";
      O;
      A     "WINCC_DB".SLIDE_GATE_3_CLOSE_STA;
      AN    "CD_OR_PC_SEL";
      );
      =     "OVEN_CHARGING_DB".SL_GT_3_CLS_STA_PB;
      A     L 0.0;
      A(;
      A     "SLIDE_GATE_3_OPN_STA";
      A     "CD_OR_PC_SEL";
      O;
      A     "WINCC_DB".SLIDE_GATE_3_OPEN_STA;
      AN    "CD_OR_PC_SEL";
      );
      =     "OVEN_CHARGING_DB".SL_GT_3_OPN_STA_PB;
      A     L 0.0;
      A     "SLIDE_GATE_1_FWD_LS";
      =     "OVEN_CHARGING_DB".SL_GT_1_CLS_LS;
      A     L 0.0;
      A     "SLIDE_GATE_1_RET_LS";
      =     "OVEN_CHARGING_DB".SL_GT_1_OPN_LS;
      A     L 0.0;
      A     "SLIDE_GATE_2_FWD_LS";
      =     "OVEN_CHARGING_DB".SL_GT_2_CLS_LS;
      A     L 0.0;
      A     "SLIDE_GATE_2_RET_LS";
      =     "OVEN_CHARGING_DB".SL_GT_2_OPN_LS;
      A     L 0.0;
      A     "SLIDE_GATE_3_FWD_LS";
      =     "OVEN_CHARGING_DB".SL_GT_3_CLS_LS;
      A     L 0.0;
      A     "SLIDE_GATE_3_REV_LS";
      =     "OVEN_CHARGING_DB".SL_GT_3_OPN_LS;
      A     L 0.0;
      A(;
      A     "OVEN_CHARGING_PB";
      A     "CD_OR_PC_SEL";
      O;
      A     "WINCC_DB".SF_1_LT_OVEN_CHARGE_STA;
      AN    "CD_OR_PC_SEL";
      );
      =     "OVEN_CHARGING_DB".OVEN_CHARGING_PB;
      A     L 0.0;
      A(;
      A     "FINISH_CHARGING";
      A     "CD_OR_PC_SEL";
      O;
      A     "WINCC_DB".FINISH_CHARGE_PB;
      AN    "CD_OR_PC_SEL";
      );
      =     "08_LID_MECHANISM_DB".FIN_CHARGE_PB;
      A     L 0.0;
      A     "PROX_MODE_SEL_SF_1";
      =     "OVEN_CHARGING_DB".SF1_ENCODE_PROXI_MODE;
      A     L 0.0;
      A     "PROX_MODE_SEL_SF_2";
      =     "OVEN_CHARGING_DB".SF2_ENCODE_PROXI_MODE;
      A     L 0.0;
      A     "PROX_MODE_SEL_SF_3";
      =     "OVEN_CHARGING_DB".SF3_ENCODE_PROXI_MODE;
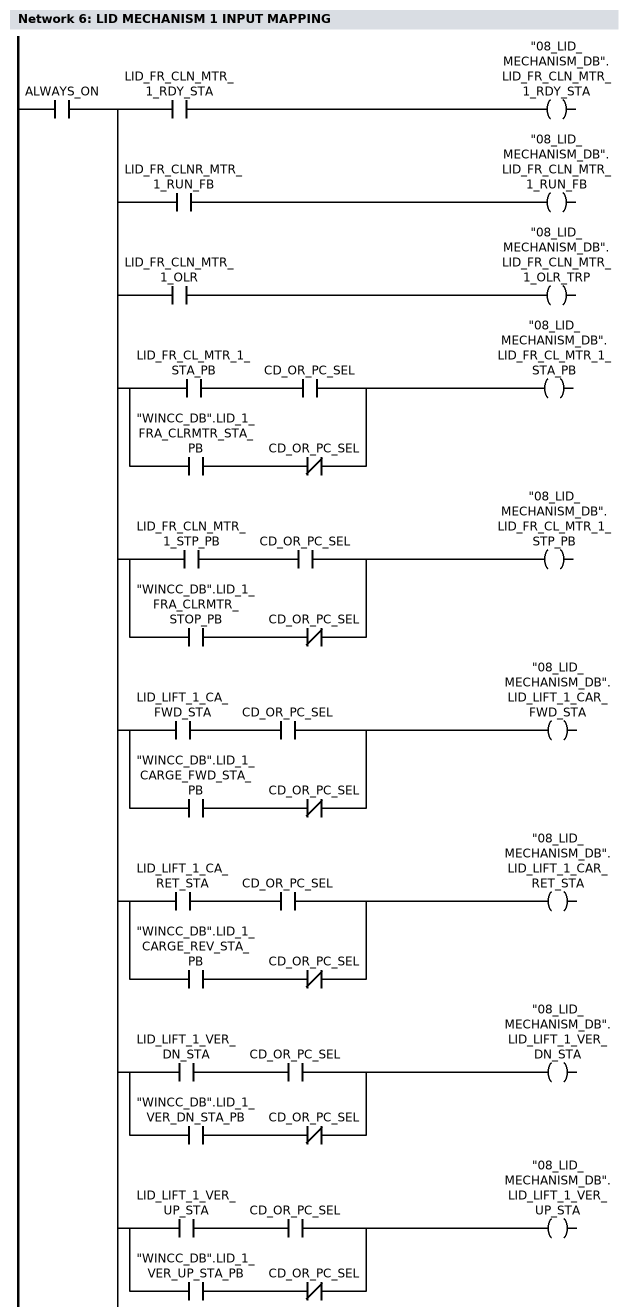
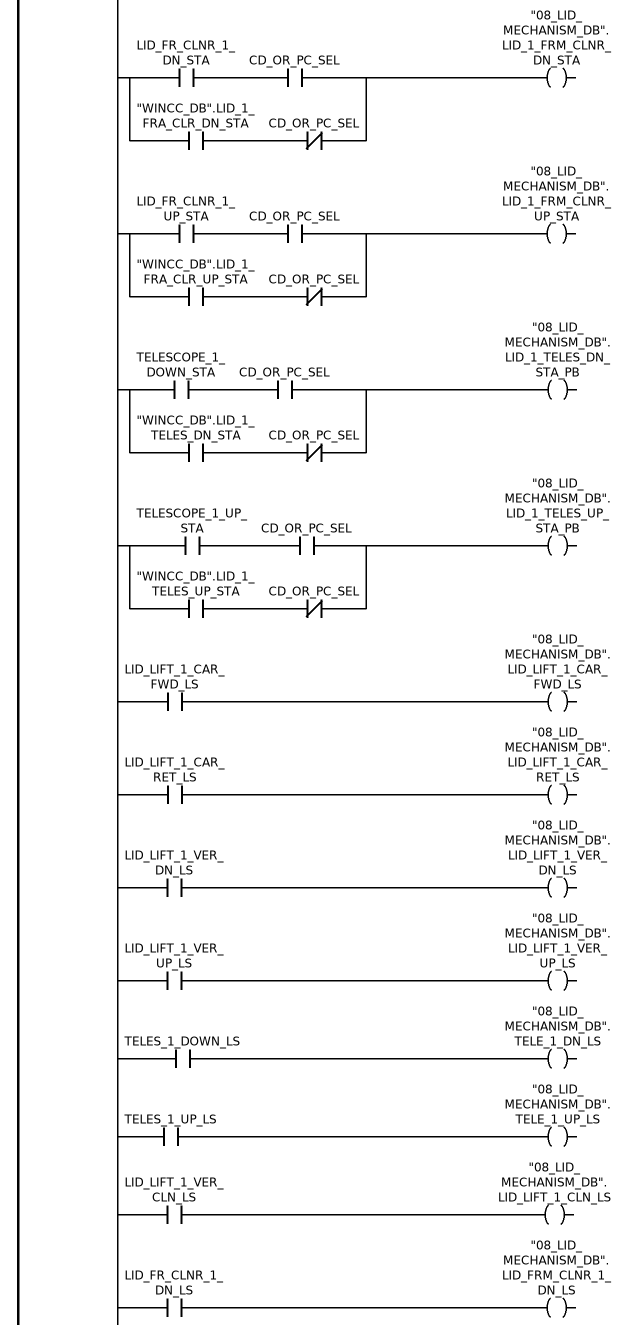
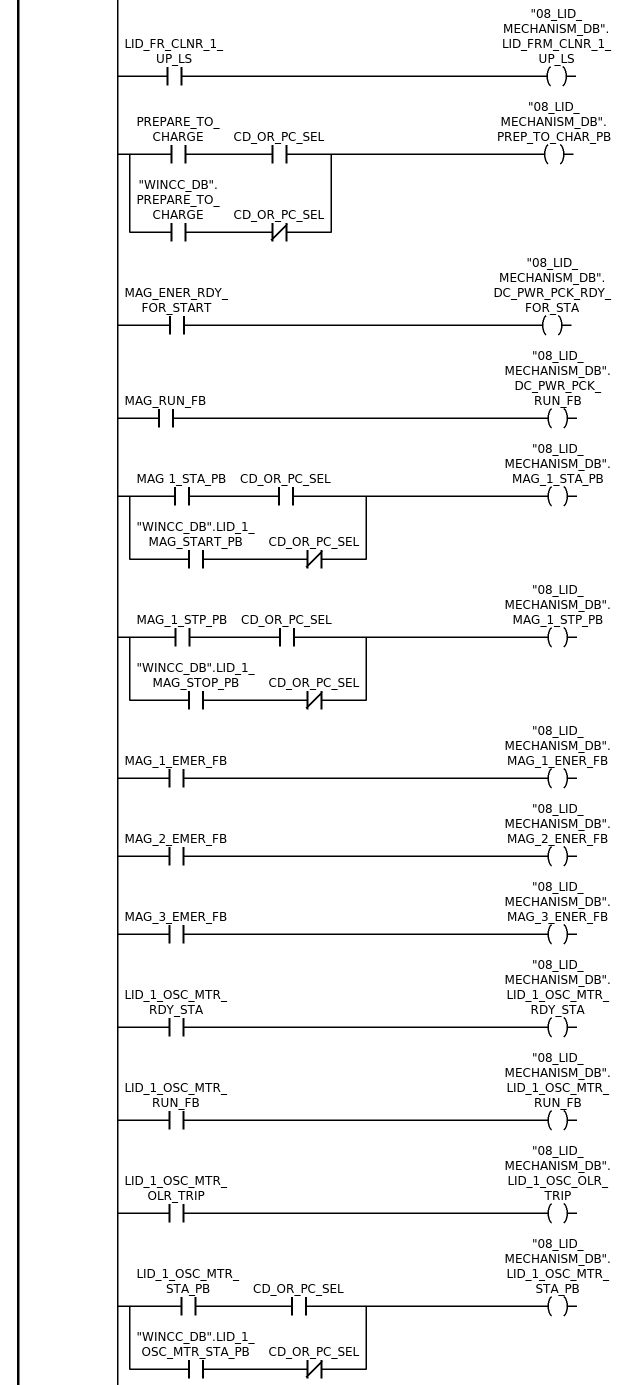
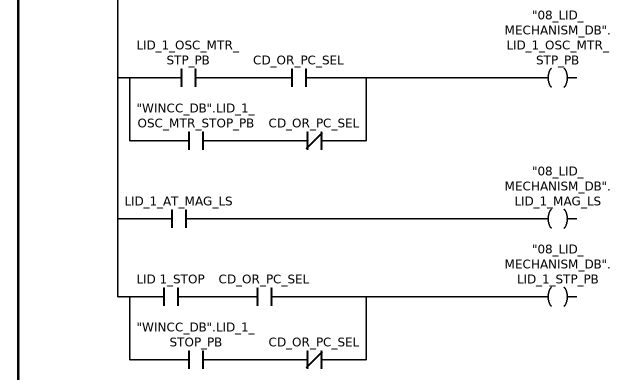
NETWORK
TITLE = LID MECHANISM 1 INPUT MAPPING
      A     "ALWAYS_ON";
      =     L 0.0;
      A     L 0.0;
      A     "LID_FR_CLN_MTR_1_RDY_STA";
      =     "08_LID_MECHANISM_DB".LID_FR_CLN_MTR_1_RDY_STA;
      A     L 0.0;
      A     "LID_FR_CLNR_MTR_1_RUN_FB";
      =     "08_LID_MECHANISM_DB".LID_FR_CLN_MTR_1_RUN_FB;
      A     L 0.0;
      A     "LID_FR_CLN_MTR_1_OLR";
      =     "08_LID_MECHANISM_DB".LID_FR_CLN_MTR_1_OLR_TRP;
      A     L 0.0;
      A(;
      A     "LID_FR_CL_MTR_1_STA_PB";
      A     "CD_OR_PC_SEL";
      O;
      A     "WINCC_DB".LID_1_FRA_CLRMTR_STA_PB;
      AN    "CD_OR_PC_SEL";
      );
      =     "08_LID_MECHANISM_DB".LID_FR_CL_MTR_1_STA_PB;
      A     L 0.0;
      A(;
      A     "LID_FR_CLN_MTR_1_STP_PB";
      A     "CD_OR_PC_SEL";
      O;
      A     "WINCC_DB".LID_1_FRA_CLRMTR_STOP_PB;
      AN    "CD_OR_PC_SEL";
      );
      =     "08_LID_MECHANISM_DB".LID_FR_CL_MTR_1_STP_PB;
      A     L 0.0;
      A(;
      A     "LID_LIFT_1_CA_FWD_STA";
      A     "CD_OR_PC_SEL";
      O;
      A     "WINCC_DB".LID_1_CARGE_FWD_STA_PB;
      AN    "CD_OR_PC_SEL";
      );
      =     "08_LID_MECHANISM_DB".LID_LIFT_1_CAR_FWD_STA;
      A     L 0.0;
      A(;
      A     "LID_LIFT_1_CA_RET_STA";
      A     "CD_OR_PC_SEL";
      O;
      A     "WINCC_DB".LID_1_CARGE_REV_STA_PB;
      AN    "CD_OR_PC_SEL";
      );
      =     "08_LID_MECHANISM_DB".LID_LIFT_1_CAR_RET_STA;
      A     L 0.0;
      A(;
      A     "LID_LIFT_1_VER_DN_STA";
      A     "CD_OR_PC_SEL";
      O;
      A     "WINCC_DB".LID_1_VER_DN_STA_PB;
      AN    "CD_OR_PC_SEL";
      );
      =     "08_LID_MECHANISM_DB".LID_LIFT_1_VER_DN_STA;
      A     L 0.0;
      A(;
      A     "LID_LIFT_1_VER_UP_STA";
      A     "CD_OR_PC_SEL";
      O;
      A     "WINCC_DB".LID_1_VER_UP_STA_PB;
      AN    "CD_OR_PC_SEL";
      );
      =     "08_LID_MECHANISM_DB".LID_LIFT_1_VER_UP_STA;
      A     L 0.0;
      A(;
      A     "LID_FR_CLNR_1_DN_STA";
      A     "CD_OR_PC_SEL";
      O;
      A     "WINCC_DB".LID_1_FRA_CLR_DN_STA;
      AN    "CD_OR_PC_SEL";
      );
      =     "08_LID_MECHANISM_DB".LID_1_FRM_CLNR_DN_STA;
      A     L 0.0;
      A(;
      A     "LID_FR_CLNR_1_UP_STA";
      A     "CD_OR_PC_SEL";
      O;
      A     "WINCC_DB".LID_1_FRA_CLR_UP_STA;
      AN    "CD_OR_PC_SEL";
      );
      =     "08_LID_MECHANISM_DB".LID_1_FRM_CLNR_UP_STA;
      A     L 0.0;
      A(;
      A     "TELESCOPE_1_DOWN_STA";
      A     "CD_OR_PC_SEL";
      O;
      A     "WINCC_DB".LID_1_TELES_DN_STA;
      AN    "CD_OR_PC_SEL";
      );
      =     "08_LID_MECHANISM_DB".LID_1_TELES_DN_STA_PB;
      A     L 0.0;
      A(;
      A     "TELESCOPE_1_UP_STA";
      A     "CD_OR_PC_SEL";
      O;
      A     "WINCC_DB".LID_1_TELES_UP_STA;
      AN    "CD_OR_PC_SEL";
      );
      =     "08_LID_MECHANISM_DB".LID_1_TELES_UP_STA_PB;
      A     L 0.0;
      A     "LID_LIFT_1_CAR_FWD_LS";
      =     "08_LID_MECHANISM_DB".LID_LIFT_1_CAR_FWD_LS;
      A     L 0.0;
      A     "LID_LIFT_1_CAR_RET_LS";
      =     "08_LID_MECHANISM_DB".LID_LIFT_1_CAR_RET_LS;
      A     L 0.0;
      A     "LID_LIFT_1_VER_DN_LS";
      =     "08_LID_MECHANISM_DB".LID_LIFT_1_VER_DN_LS;
      A     L 0.0;
      A     "LID_LIFT_1_VER_UP_LS";
      =     "08_LID_MECHANISM_DB".LID_LIFT_1_VER_UP_LS;
      A     L 0.0;
      A     "TELES_1_DOWN_LS";
      =     "08_LID_MECHANISM_DB".TELE_1_DN_LS;
      A     L 0.0;
      A     "TELES_1_UP_LS";
      =     "08_LID_MECHANISM_DB".TELE_1_UP_LS;
      A     L 0.0;
      A     "LID_LIFT_1_VER_CLN_LS";
      =     "08_LID_MECHANISM_DB".LID_LIFT_1_CLN_LS;
      A     L 0.0;
      A     "LID_FR_CLNR_1_DN_LS";
      =     "08_LID_MECHANISM_DB".LID_FRM_CLNR_1_DN_LS;
      A     L 0.0;
      A     "LID_FR_CLNR_1_UP_LS";
      =     "08_LID_MECHANISM_DB".LID_FRM_CLNR_1_UP_LS;
      A     L 0.0;
      A(;
      A     "PREPARE_TO_CHARGE";
      A     "CD_OR_PC_SEL";
      O;
      A     "WINCC_DB".PREPARE_TO_CHARGE;
      AN    "CD_OR_PC_SEL";
      );
      =     "08_LID_MECHANISM_DB".PREP_TO_CHAR_PB;
      A     L 0.0;
      A     "MAG_ENER_RDY_FOR_START";
      =     "08_LID_MECHANISM_DB".DC_PWR_PCK_RDY_FOR_STA;
      A     L 0.0;
      A     "MAG_RUN_FB";
      =     "08_LID_MECHANISM_DB".DC_PWR_PCK_RUN_FB;
      A     L 0.0;
      A(;
      A     "MAG 1_STA_PB";
      A     "CD_OR_PC_SEL";
      O;
      A     "WINCC_DB".LID_1_MAG_START_PB;
      AN    "CD_OR_PC_SEL";
      );
      =     "08_LID_MECHANISM_DB".MAG_1_STA_PB;
      A     L 0.0;
      A(;
      A     "MAG_1_STP_PB";
      A     "CD_OR_PC_SEL";
      O;
      A     "WINCC_DB".LID_1_MAG_STOP_PB;
      AN    "CD_OR_PC_SEL";
      );
      =     "08_LID_MECHANISM_DB".MAG_1_STP_PB;
      A     L 0.0;
      A     "MAG_1_EMER_FB";
      =     "08_LID_MECHANISM_DB".MAG_1_ENER_FB;
      A     L 0.0;
      A     "MAG_2_EMER_FB";
      =     "08_LID_MECHANISM_DB".MAG_2_ENER_FB;
      A     L 0.0;
      A     "MAG_3_EMER_FB";
      =     "08_LID_MECHANISM_DB".MAG_3_ENER_FB;
      A     L 0.0;
      A     "LID_1_OSC_MTR_RDY_STA";
      =     "08_LID_MECHANISM_DB".LID_1_OSC_MTR_RDY_STA;
      A     L 0.0;
      A     "LID_1_OSC_MTR_RUN_FB";
      =     "08_LID_MECHANISM_DB".LID_1_OSC_MTR_RUN_FB;
      A     L 0.0;
      A     "LID_1_OSC_MTR_OLR_TRIP";
      =     "08_LID_MECHANISM_DB".LID_1_OSC_OLR_TRIP;
      A     L 0.0;
      A(;
      A     "LID_1_OSC_MTR_STA_PB";
      A     "CD_OR_PC_SEL";
      O;
      A     "WINCC_DB".LID_1_OSC_MTR_STA_PB;
      AN    "CD_OR_PC_SEL";
      );
      =     "08_LID_MECHANISM_DB".LID_1_OSC_MTR_STA_PB;
      A     L 0.0;
      A(;
      A     "LID_1_OSC_MTR_STP_PB";
      A     "CD_OR_PC_SEL";
      O;
      A     "WINCC_DB".LID_1_OSC_MTR_STOP_PB;
      AN    "CD_OR_PC_SEL";
      );
      =     "08_LID_MECHANISM_DB".LID_1_OSC_MTR_STP_PB;
      A     L 0.0;
      A     "LID_1_AT_MAG_LS";
      =     "08_LID_MECHANISM_DB".LID_1_MAG_LS;
      A     L 0.0;
      A(;
      A     "LID 1_STOP";
      A     "CD_OR_PC_SEL";
      O;
      A     "WINCC_DB".LID_1_STOP_PB;
      AN    "CD_OR_PC_SEL";
      );
      =     "08_LID_MECHANISM_DB".LID_1_STP_PB;
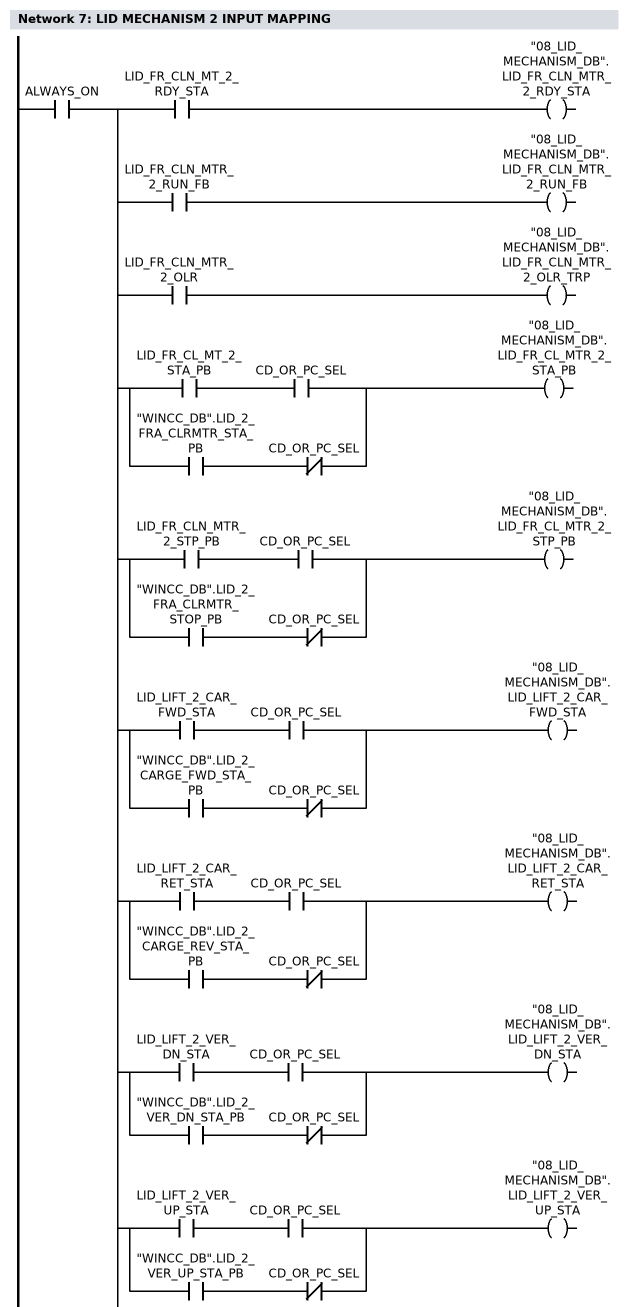
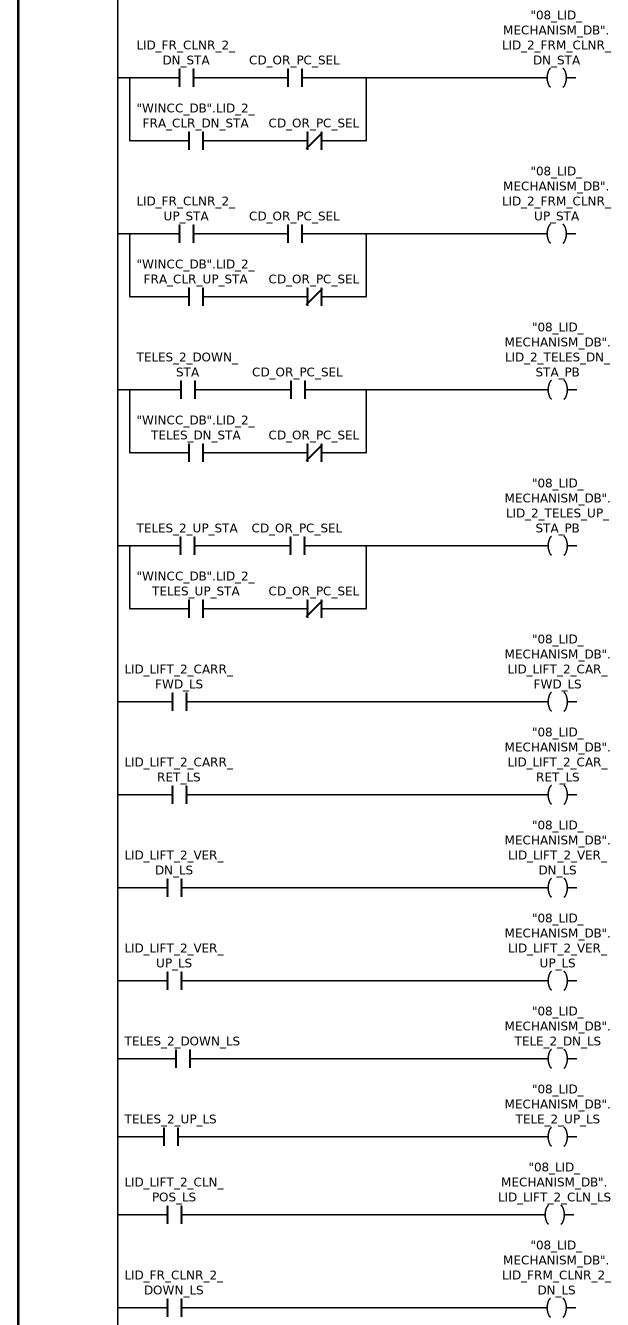
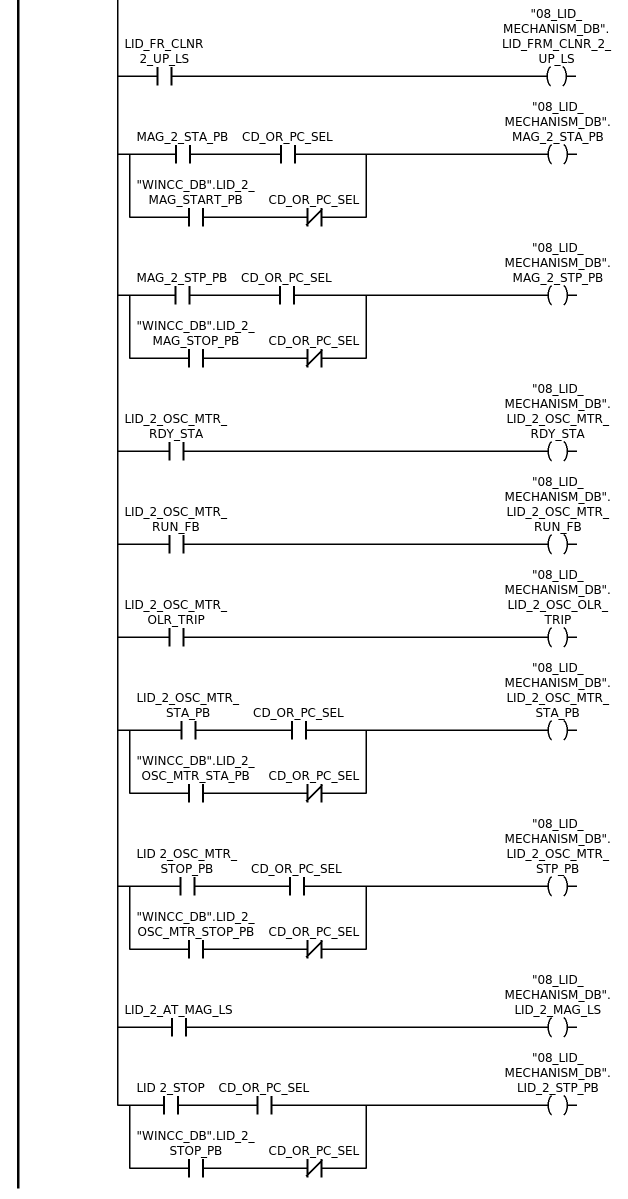
NETWORK
TITLE = LID MECHANISM 2 INPUT MAPPING
      A     "ALWAYS_ON";
      =     L 0.0;
      A     L 0.0;
      A     "LID_FR_CLN_MT_2_RDY_STA";
      =     "08_LID_MECHANISM_DB".LID_FR_CLN_MTR_2_RDY_STA;
      A     L 0.0;
      A     "LID_FR_CLN_MTR_2_RUN_FB";
      =     "08_LID_MECHANISM_DB".LID_FR_CLN_MTR_2_RUN_FB;
      A     L 0.0;
      A     "LID_FR_CLN_MTR_2_OLR";
      =     "08_LID_MECHANISM_DB".LID_FR_CLN_MTR_2_OLR_TRP;
      A     L 0.0;
      A(;
      A     "LID_FR_CL_MT_2_STA_PB";
      A     "CD_OR_PC_SEL";
      O;
      A     "WINCC_DB".LID_2_FRA_CLRMTR_STA_PB;
      AN    "CD_OR_PC_SEL";
      );
      =     "08_LID_MECHANISM_DB".LID_FR_CL_MTR_2_STA_PB;
      A     L 0.0;
      A(;
      A     "LID_FR_CLN_MTR_2_STP_PB";
      A     "CD_OR_PC_SEL";
      O;
      A     "WINCC_DB".LID_2_FRA_CLRMTR_STOP_PB;
      AN    "CD_OR_PC_SEL";
      );
      =     "08_LID_MECHANISM_DB".LID_FR_CL_MTR_2_STP_PB;
      A     L 0.0;
      A(;
      A     "LID_LIFT_2_CAR_FWD_STA";
      A     "CD_OR_PC_SEL";
      O;
      A     "WINCC_DB".LID_2_CARGE_FWD_STA_PB;
      AN    "CD_OR_PC_SEL";
      );
      =     "08_LID_MECHANISM_DB".LID_LIFT_2_CAR_FWD_STA;
      A     L 0.0;
      A(;
      A     "LID_LIFT_2_CAR_RET_STA";
      A     "CD_OR_PC_SEL";
      O;
      A     "WINCC_DB".LID_2_CARGE_REV_STA_PB;
      AN    "CD_OR_PC_SEL";
      );
      =     "08_LID_MECHANISM_DB".LID_LIFT_2_CAR_RET_STA;
      A     L 0.0;
      A(;
      A     "LID_LIFT_2_VER_DN_STA";
      A     "CD_OR_PC_SEL";
      O;
      A     "WINCC_DB".LID_2_VER_DN_STA_PB;
      AN    "CD_OR_PC_SEL";
      );
      =     "08_LID_MECHANISM_DB".LID_LIFT_2_VER_DN_STA;
      A     L 0.0;
      A(;
      A     "LID_LIFT_2_VER_UP_STA";
      A     "CD_OR_PC_SEL";
      O;
      A     "WINCC_DB".LID_2_VER_UP_STA_PB;
      AN    "CD_OR_PC_SEL";
      );
      =     "08_LID_MECHANISM_DB".LID_LIFT_2_VER_UP_STA;
      A     L 0.0;
      A(;
      A     "LID_FR_CLNR_2_DN_STA";
      A     "CD_OR_PC_SEL";
      O;
      A     "WINCC_DB".LID_2_FRA_CLR_DN_STA;
      AN    "CD_OR_PC_SEL";
      );
      =     "08_LID_MECHANISM_DB".LID_2_FRM_CLNR_DN_STA;
      A     L 0.0;
      A(;
      A     "LID_FR_CLNR_2_UP_STA";
      A     "CD_OR_PC_SEL";
      O;
      A     "WINCC_DB".LID_2_FRA_CLR_UP_STA;
      AN    "CD_OR_PC_SEL";
      );
      =     "08_LID_MECHANISM_DB".LID_2_FRM_CLNR_UP_STA;
      A     L 0.0;
      A(;
      A     "TELES_2_DOWN_STA";
      A     "CD_OR_PC_SEL";
      O;
      A     "WINCC_DB".LID_2_TELES_DN_STA;
      AN    "CD_OR_PC_SEL";
      );
      =     "08_LID_MECHANISM_DB".LID_2_TELES_DN_STA_PB;
      A     L 0.0;
      A(;
      A     "TELES_2_UP_STA";
      A     "CD_OR_PC_SEL";
      O;
      A     "WINCC_DB".LID_2_TELES_UP_STA;
      AN    "CD_OR_PC_SEL";
      );
      =     "08_LID_MECHANISM_DB".LID_2_TELES_UP_STA_PB;
      A     L 0.0;
      A     "LID_LIFT_2_CARR_FWD_LS";
      =     "08_LID_MECHANISM_DB".LID_LIFT_2_CAR_FWD_LS;
      A     L 0.0;
      A     "LID_LIFT_2_CARR_RET_LS";
      =     "08_LID_MECHANISM_DB".LID_LIFT_2_CAR_RET_LS;
      A     L 0.0;
      A     "LID_LIFT_2_VER_DN_LS";
      =     "08_LID_MECHANISM_DB".LID_LIFT_2_VER_DN_LS;
      A     L 0.0;
      A     "LID_LIFT_2_VER_UP_LS";
      =     "08_LID_MECHANISM_DB".LID_LIFT_2_VER_UP_LS;
      A     L 0.0;
      A     "TELES_2_DOWN_LS";
      =     "08_LID_MECHANISM_DB".TELE_2_DN_LS;
      A     L 0.0;
      A     "TELES_2_UP_LS";
      =     "08_LID_MECHANISM_DB".TELE_2_UP_LS;
      A     L 0.0;
      A     "LID_LIFT_2_CLN_POS_LS";
      =     "08_LID_MECHANISM_DB".LID_LIFT_2_CLN_LS;
      A     L 0.0;
      A     "LID_FR_CLNR_2_DOWN_LS";
      =     "08_LID_MECHANISM_DB".LID_FRM_CLNR_2_DN_LS;
      A     L 0.0;
      A     "LID_FR_CLNR 2_UP_LS";
      =     "08_LID_MECHANISM_DB".LID_FRM_CLNR_2_UP_LS;
      A     L 0.0;
      A(;
      A     "MAG_2_STA_PB";
      A     "CD_OR_PC_SEL";
      O;
      A     "WINCC_DB".LID_2_MAG_START_PB;
      AN    "CD_OR_PC_SEL";
      );
      =     "08_LID_MECHANISM_DB".MAG_2_STA_PB;
      A     L 0.0;
      A(;
      A     "MAG_2_STP_PB";
      A     "CD_OR_PC_SEL";
      O;
      A     "WINCC_DB".LID_2_MAG_STOP_PB;
      AN    "CD_OR_PC_SEL";
      );
      =     "08_LID_MECHANISM_DB".MAG_2_STP_PB;
      A     L 0.0;
      A     "LID_2_OSC_MTR_RDY_STA";
      =     "08_LID_MECHANISM_DB".LID_2_OSC_MTR_RDY_STA;
      A     L 0.0;
      A     "LID_2_OSC_MTR_RUN_FB";
      =     "08_LID_MECHANISM_DB".LID_2_OSC_MTR_RUN_FB;
      A     L 0.0;
      A     "LID_2_OSC_MTR_OLR_TRIP";
      =     "08_LID_MECHANISM_DB".LID_2_OSC_OLR_TRIP;
      A     L 0.0;
      A(;
      A     "LID_2_OSC_MTR_STA_PB";
      A     "CD_OR_PC_SEL";
      O;
      A     "WINCC_DB".LID_2_OSC_MTR_STA_PB;
      AN    "CD_OR_PC_SEL";
      );
      =     "08_LID_MECHANISM_DB".LID_2_OSC_MTR_STA_PB;
      A     L 0.0;
      A(;
      A     "LID 2_OSC_MTR_STOP_PB";
      A     "CD_OR_PC_SEL";
      O;
      A     "WINCC_DB".LID_2_OSC_MTR_STOP_PB;
      AN    "CD_OR_PC_SEL";
      );
      =     "08_LID_MECHANISM_DB".LID_2_OSC_MTR_STP_PB;
      A     L 0.0;
      A     "LID_2_AT_MAG_LS";
      =     "08_LID_MECHANISM_DB".LID_2_MAG_LS;
      A     L 0.0;
      A(;
      A     "LID 2_STOP";
      A     "CD_OR_PC_SEL";
      O;
      A     "WINCC_DB".LID_2_STOP_PB;
      AN    "CD_OR_PC_SEL";
      );
      =     "08_LID_MECHANISM_DB".LID_2_STP_PB;
